(* CODESYS project sms_festo_lib_v1_1.library
   Company: Festo
   Description: 1.1.0 Added Intermediate Block
   Version: 1.1.0
   Placeholder: SMS Festo Lib V1.1
   Author: AJAY
   Title: SMS Festo Lib

Project tree, tasks and I/O mapping:
  libraries: Festo_CPX_API_EC_Beckhoff, * (Festo); Tc2_Standard, * (Beckhoff Automation GmbH); Tc2_System, * (Beckhoff Automation GmbH); Tc3_Module, * (Beckhoff Automation GmbH)
  DUTs/
    data type aByte_as_real
    data type UDT_ISDU_Command
    data type UDT_ReadParameter
    data type UDT_WriteParameter
  GVLs/
    global variables GVL
  POUs/
    function block SMS_Festo_Advanced [ST]
    function block SMS_Festo_Basic [ST]
    function block SMS_Festo_Intermediate [ST]
    function block SMS_Festo_IO [ST]
  Project Information/
    function F_GetCompany [ST]
    function F_GetTitle [ST]
    function F_GetVersion [ST]
  Version/
    global variables Global_Version
  VISUs/
*)

// DUTs/aByte_as_real
TYPE aByte_as_real :
UNION
	rRealValue: REAL;
	abyte: ARRAY  [0..3] OF BYTE;
END_UNION
END_TYPE

// DUTs/UDT_ISDU_Command
TYPE UDT_ISDU_Command :
STRUCT
	Net_Id: STRING;
	Ethercat_Address: 	UINT;
	Slot_Number: 	UINT;
	Port_Number: 	USINT;
	Para_Index: 	UINT;
	Para_SubIndex: 	USINT;
	Para_Length: 	UINT;
	Para_Data: 		ARRAY[0..231] OF BYTE;
	
END_STRUCT
END_TYPE

// DUTs/UDT_ReadParameter
TYPE UDT_ReadParameter :
STRUCT
	Index	:	UINT;	// Read Data Parameter Index Value
	Sub_index	:	USINT;	// Read Data Parameter Sub index Value
	Length		:	UINT;	// Read Data Parameter Length Value
	Value		:	DINT;	// Read Data Parameter Feedback Value
END_STRUCT
END_TYPE

// DUTs/UDT_WriteParameter
TYPE UDT_WriteParameter :
STRUCT
	Index		:	UINT;	// Send Data Parameter Index Value
	Sub_index		:	USINT;	// Send Data Parameter sub index Value
	Length			:	UINT;	// Send Data Parameter Length Value
	Value			:	DINT;	// Send Data Parameter Write Value
	NeedAction		:	BOOL;	// Send Data Parameter Need Action Decision 
	PreviousValue	:	DINT;	// Send Data Parameter Previous Write Value
	REAL_Value		:	REAL;	// Send Data Parameter Write REAL Value
END_STRUCT
END_TYPE

// GVLs/GVL
{attribute 'qualified_only'}
VAR_GLOBAL
	Inputs AT %I*: BYTE;
	Outputs AT %Q*: BYTE;
END_VAR

// Version/Global_Version
{attribute 'TcGenerated'}
{attribute 'no-analysis'}
{attribute 'linkalways'}
// This function has been automatically generated from the project information.
VAR_GLOBAL CONSTANT
	{attribute 'const_non_replaced'}
	stLibVersion_SMS_Festo_Lib : ST_LibVersion := (iMajor := 1, iMinor := 1, iBuild := 0, iRevision := 0, nFlags := 0, sVersion := '1.1.0');
END_VAR

// POUs/SMS_Festo_Advanced
FUNCTION_BLOCK SMS_Festo_Advanced
VAR_INPUT
	RefINPUTS: BYTE;					//Input Channel Mapping
	xEnable: BOOL; 						//True - Enable AOI function
	sNetId              : STRING;
	uiEthercatAddress   : UINT;          //Address of the slave device i.e. CPX-AP-I-EC-M12 Module
	uiSlotNumber        : UINT;          //Slot number where the IO Link master CPX-AP-I-4IOL-M12 module is connected
	usiPort             : USINT;          //Port of the CPX-AP-I-4IOL-M12 module where IO link device is connected
	xMoveIN: BOOL;						//TRUE - SMS moves inwards | FALSE - SMS Stops		
	xMoveIntermediate: BOOL;			//TRUE – SMS Moves to Intermediate Position | FALSE – SMS Stops
	xMoveOut: BOOL;						//TRUE - SMS moves outwards | FALSE - SMS Stops
	xQuitError: BOOL;					//TRUE - Reset Error Messages
	xPowerSMS: BOOL;					//TRUE - Enable power stage of SMS
	xUserInterfaceLock: BOOL;			//TRUE - lock user interface of SMS control unit
	bySpeedOut: BYTE := 1;				//Axix Move Speed Towards Out Direction 1 - 10% (default) | Limit 1 to 10
	bySpeedIN: BYTE:= 1;				//Axix Move Speed Towards IN Direction 1 - 10% (default) | Limit 1 to 10
	byForce: BYTE:= 1;					//Axix Move Force 1 - 10% (default) | Limit 1 to 10
	xReferenceDirection: BOOL;			//TRUE - Motor averted | FALSE - Motor side
	xExecuteReference: BOOL;			//TRUE – Start Homing
	diStartPressPosition: DINT:= 100;	//Defines Start Position of Stroke
	diIntermediatePosition: DINT:= 200;	//Defines Intermediate Position of Stroke
	diEndPosition: DINT:= 300;			//Defines End Position of Stroke
	xAutoStoreActive: BOOL;				//TRUE – Automatically stores the last downloaded parameters in the SMS.
	xStoreParameters: BOOL;				//TRUE – Manually stores the last downloaded parameters in the SMS.
	xReadDiagnosticData: BOOL;			//TRUE - Update value of outputs: O_DDTemperature, O_DDCurrent, O_DDVoltage, O_DDCyclesTotal, O_DDCyclesSinceReset, O_DDMileageTotal, O_DDMileageSinceReset
	xResetCounterMileage: BOOL;			//TRUE - Resets values of parameters “O_DDCyclesSinceReset”
	
END_VAR
VAR_OUTPUT
	RefOUTPUTS: BYTE;					//Output Channel Mapping
	xEnabled: BOOL;						//TRUE - AOI Function Enabled
	xWriteActive: BOOL;					//TRUE - Executing Parameter Write Function
	xWriteDone: BOOL;					//TRUE - Last Parameter Wrote Successful
	xReadActive: BOOL;					//TRUE - Parameter Read Function is Active
	xStateIn: BOOL;						//TRUE - SMS Axis Reached IN Position
	xStateIntermediate: BOOL;			//TRUE - SMS Axis Reached Intermediate Position
	xStateOut: BOOL;					//TRUE - SMS Axis Reached OUT Position
	xStateMove: BOOL;					//TRUE – SMS Axis at Moving Condition | FALSE – SMS Axis at Ideal Condition
	xError: BOOL;						//TRUE - SMS Module or AOI in Error State. Check Error Code
	uiLocalError: UINT;					//Function Block Local Error Code
	aErrorCode: ARRAY[0..15] OF WORD;	//SMS Error Code List
	diCurrentPosition: DINT;			//Axis Current Position Feedback
	diCurrentSpeed: DINT;				//Axis Current Speed Feedback
	diCurrentForce: DINT;				//Axis Current Force Feedback
	diDDTemprature: DINT;				//SMS Module Current Temperature Feedback
	diDDCurrent: DINT;					//SMS Module Present Value of Current
	diDDVoltage: DINT;					//SMS Module Present Voltage Feedback
	diDDCyclesTotal: DINT;				//Sum Value of Total Number of Axis Movement Cycle Count
	diDDCyclesSinceReset: DINT;			//Number of Axis Movement Cycle Count Since Reset Command
	diDDMileageTotal: DINT;				//Total Number of Movement Cycle in Engineering Unit
	diDDMileagesSinceReset: DINT;		//Number of Axis Movement Engineered Value Since Reset Command
	diNumOfStorageOperation: DINT;		//Total Number of Auto Store Operation Done Sofare
	
END_VAR

VAR
	Lt_ReadParaData: ARRAY[0..19] OF UDT_ReadParameter;
	Lt_WriteParaData: ARRAY[0..19] OF UDT_WriteParameter;
	Lt_ErrorRawData: ARRAY [0..48] OF BYTE;
	Lt_RiseEdgePowerSMS: BOOL;
	Lt_FalingEdgePowerSMS: BOOL;
	Lt_RiseUserInterfaceLock: BOOL;
	Lt_FalingEdgeUserInterfaceLock: BOOL;
	Lt_RiseReferenceDirection: BOOL;
	Lt_FalingEdgeReferenceDirection: BOOL;
	Lt_RiseExecuteReference: BOOL;
	Lt_FalingEdgeExecuteReference: BOOL;
	Lt_RiseStoreParameters: BOOL;
	Lt_FalingEdgeStoreParameters: BOOL;
	Lt_RiseResetCounterMileage: BOOL;
	Lt_FalingEdgeResetCounterMileage: BOOL;
	Lt_RiseAutoStoreActive: BOOL;
	Lt_FalingEdgeAutoStoreActive: BOOL;
	Lt_RiseEnableFileHandling: BOOL;
	Lt_FalingEdgeEnableFileHandling: BOOL;
	Step_SEQ: INT;
	Lt_ReadIndex: INT;
	Lt_WriteIndex: INT;
	Lt_Read_Parameter_ISDU: UDT_ISDU_Command;
	Lt_Write_Parameter_ISDU: UDT_ISDU_Command;
	Lt_ForLength: INT;
	Lt_Execute_Read: BOOL;
	Lt_Execute_Write: BOOL; 
	Lt_StateDevice: BOOL;
	Lt_ScanCount: DINT;
	Lt_ScanCount02: DINT;
	Lt_ScanCount03: DINT;
	Lt_ScanCount001: DINT;
	Lt_DeviceState_RisingEdge: BOOL;
	Lt_RealConvert: aByte_as_real;
	Lt_ExecuteReference_RisingEdge: BOOL;
	Lt_ExecuteReference_Trigger: BOOL;
	Lt_ExecuteReference_Trigger01: BOOL;	
	Lt_IsItString: BOOL;
	Lt_Startposition: REAL;
	Lt_Intermediateposition: REAL;
	Lt_Endposition: REAL;
	Lt_ReCurrentPosition: REAL;
	Lt_ReCurrentPosition1: DINT;
	LT_ParameterRewriteDelay: BOOL;
	Lt_ExecuteReference_Trigger02: BOOL;
	Lt_NumOfStorageOperation:Dint;
	
	ReadPara: CPXAPI_IOLink_Parameter;
	WritePara: CPXAPI_IOLink_Parameter;
	Delay_Timmer: TON;
	Elapse_time: TIME;
END_VAR

(*
fkjhfkjsdhjkfhsdjkfhkjhhh
jdhfjkdhjkfhdkjhf
*)

(*
===============================================================================================================
Advice TO Released Library Revisions 
===============================================================================================================
SMS_Festo_Lib | Communication: Beckhoff EtherCat
---------------------------------------------------------------------------------------------------------------
Version                           Date of Release
V1.0                                07.01.2022
V1.1                                03.06.2022

---------------------------------------------------------------------------------------------------------------
Changes in Library:

V1.0 -  Release Version


V1.1 - Position variables datatype changed from Real to Dint.
       Autostorage parameter continuous count bug fixed.
       Number of storage parameter double count bug fixed. 
*)

// Enable Function Block Sequence Logic------------------------------------------------------------------------ 
IF xEnable THEN 				
	xEnabled					:= TRUE;
	
ELSE
	xEnabled					:= FALSE;
	xWriteActive				:= FALSE;	
	xWriteDone					:= FALSE;
	xReadActive					:= FALSE;
	Step_SEQ					:= 0;
	Lt_ReadParaData[0].Value	:= 0;
	Lt_ReadParaData[1].Value	:= 0;
	Lt_ReadParaData[2].Value	:= 0;
	Lt_ReadParaData[3].Value	:= 0;
	Lt_ReadParaData[4].Value	:= 0;
	Lt_ReadParaData[5].Value	:= 0;
	Lt_ReadParaData[6].Value	:= 0;
	Lt_ReadParaData[7].Value	:= 0;
	Lt_ReadParaData[8].Value	:= 0;
	Lt_ReadParaData[9].Value	:= 0;
	Lt_ReadParaData[10].Value	:= 0;
	Lt_ReadParaData[11].Value	:= 0;
	
END_IF

//Process Data Command Logic---------------------------------------------------------------------------------------
IF xEnabled THEN				
	
	IF xMoveIN THEN				// Move IN Position Command
		RefOUTPUTS.0	:= TRUE;
	ELSE
		RefOUTPUTS.0	:= FALSE;
	END_IF
	
	IF xMoveOut THEN			// Move OUT Position Command
		RefOUTPUTS.1	:= TRUE;
	ELSE
		RefOUTPUTS.1	:= FALSE;	
	END_IF
	
	IF xMoveIntermediate THEN	// Move Intermediat Position Command
		RefOUTPUTS.4	:= TRUE;
	ELSE
		RefOUTPUTS.4	:= FALSE;	
	END_IF
	
	IF xQuitError THEN			// Move Quite Error Command
		RefOUTPUTS.2	:= TRUE;
	ELSE
		RefOUTPUTS.2	:= FALSE;	
	END_IF
ELSE							// Clear Command When FB Not Enabled
	RefOUTPUTS.0	:= FALSE;	
	RefOUTPUTS.1	:= FALSE;	
	RefOUTPUTS.2	:= FALSE;
	RefOUTPUTS.4	:= FALSE;
END_IF


// Process Data Feedback Logic---------------------------------------------------------------------------------
IF xEnabled THEN				
	
	IF RefINPUTS.0 THEN				// IN Position Status
		xStateIn	:= TRUE;
	ELSE
		xStateIn	:= FALSE;
	END_IF
	
	IF RefINPUTS.1 THEN				// Out Position Status
		xStateOut	:= TRUE;
	ELSE
		xStateOut	:= FALSE;
	END_IF
	
	IF RefINPUTS.2 THEN				// Axis Moving Status
		xStateMove	:= TRUE;
	ELSE
		xStateMove	:= FALSE;
	END_IF
	
	IF RefINPUTS.3 THEN				// Device Healthy Status
		Lt_StateDevice	:= TRUE;
	ELSE
		Lt_StateDevice	:= FALSE;
	END_IF
	
	IF RefINPUTS.4 THEN				// Intermediat Position Status
		xStateIntermediate	:= TRUE;
	ELSE
		xStateIntermediate	:= FALSE;
	END_IF	
ELSE 								// Clear Status When FB is Not Enabled
	xStateIn			:= FALSE;
	xStateOut			:= FALSE;
	xStateMove			:= FALSE;
	xStateIntermediate	:= FALSE;
	Lt_StateDevice		:= FALSE;
END_IF

// Device Error State Logic -----------------------------------------------------------------------------------
IF xEnabled AND xStateIn AND xStateOut AND NOT Lt_StateDevice THEN
	xError	:= TRUE;
ELSE
	xError	:= FALSE;
END_IF

// After Homing Parameters Re-Write Logic ---------------------------------------------------------------------
IF Lt_ExecuteReference_Trigger01	AND NOT xStateMove THEN
	Lt_ExecuteReference_Trigger02:= TRUE;
	
	IF LT_ParameterRewriteDelay THEN
		Lt_WriteParaData[0].PreviousValue	:= 0;
		Lt_WriteParaData[1].PreviousValue	:= 0;
		Lt_WriteParaData[2].PreviousValue	:= 0;
		Lt_WriteParaData[3].PreviousValue	:= 0;
		Lt_WriteParaData[4].PreviousValue	:= 0;
		Lt_WriteParaData[5].PreviousValue	:= 0;
		Lt_WriteParaData[7].PreviousValue	:= 0;
		Lt_WriteParaData[8].PreviousValue	:= 0;
		Lt_WriteParaData[12].PreviousValue	:= 0;
		Lt_ExecuteReference_Trigger01		:= FALSE;
		Lt_ExecuteReference_Trigger02		:= FALSE;
		
	END_IF
ELSE
		Lt_ExecuteReference_Trigger02		:= FALSE;
END_IF
// After Homing Parameter Rewrite Delay
Delay_Timmer(IN:= Lt_ExecuteReference_Trigger02, PT:=T#6S , Q=> LT_ParameterRewriteDelay, ET=> Elapse_time );

//Setpoint Limit Error-----------------------------------------------------------------------------------------
IF (bySpeedIN < 1 ) OR (bySpeedIN > 10 ) THEN 
	uiLocalError := 1001;
	xError		 := TRUE;

ELSIF (bySpeedOut < 1 ) OR (bySpeedOut > 10 ) THEN
	uiLocalError := 1002;
	xError		 := TRUE;
ELSIF (bySpeedIN < 1 ) OR (bySpeedIN > 10 ) THEN
	uiLocalError := 1003;
	xError		 := TRUE;
END_IF

//Device Status Rising Edge Logic--------------------------------------------------------------------------------
IF Lt_StateDevice AND NOT Lt_DeviceState_RisingEdge THEN
	Lt_DeviceState_RisingEdge	:= TRUE;
	xError						:= FALSE;
ELSIF NOT Lt_StateDevice THEN
	Lt_DeviceState_RisingEdge	:= FALSE;
END_IF

//Execute Ref Rising Edge Logic--------------------------------------------------------------------------------
IF xExecuteReference AND NOT Lt_ExecuteReference_RisingEdge THEN
	Lt_ExecuteReference_RisingEdge	:= TRUE;
	Lt_ExecuteReference_Trigger		:= TRUE;
	xError							:= FALSE;
ELSIF NOT xExecuteReference THEN
	Lt_ExecuteReference_RisingEdge	:= FALSE;
END_IF

// Quite Error Logic ------------------------------------------------------------------------------------------
IF xQuitError AND xEnabled THEN
	Step_SEQ			:= 0;
	xWriteActive		:= FALSE;
	xWriteDone			:= FALSE;
	xReadActive			:= FALSE;
	xError				:= FALSE;
	uiLocalError		:= 0;	
	
	// Clear Error Data Raw Array
		
				Lt_ErrorRawData[0] 		:= 0; Lt_ErrorRawData[1] 	:= 0; Lt_ErrorRawData[2] 	:= 0; Lt_ErrorRawData[3] 	:= 0;
				Lt_ErrorRawData[4] 		:= 0; Lt_ErrorRawData[5] 	:= 0; Lt_ErrorRawData[6] 	:= 0; Lt_ErrorRawData[7] 	:= 0;
				Lt_ErrorRawData[8] 		:= 0; Lt_ErrorRawData[9] 	:= 0; Lt_ErrorRawData[10] 	:= 0; Lt_ErrorRawData[11] 	:= 0;
				Lt_ErrorRawData[12] 	:= 0; Lt_ErrorRawData[13] 	:= 0; Lt_ErrorRawData[14] 	:= 0; Lt_ErrorRawData[15] 	:= 0;
				Lt_ErrorRawData[16] 	:= 0; Lt_ErrorRawData[17] 	:= 0; Lt_ErrorRawData[18] 	:= 0; Lt_ErrorRawData[19] 	:= 0;
				Lt_ErrorRawData[20] 	:= 0; Lt_ErrorRawData[21] 	:= 0; Lt_ErrorRawData[22] 	:= 0; Lt_ErrorRawData[23] 	:= 0;
				Lt_ErrorRawData[24] 	:= 0; Lt_ErrorRawData[25] 	:= 0; Lt_ErrorRawData[26] 	:= 0; Lt_ErrorRawData[27] 	:= 0;
				Lt_ErrorRawData[28] 	:= 0; Lt_ErrorRawData[29] 	:= 0; Lt_ErrorRawData[30] 	:= 0; Lt_ErrorRawData[31] 	:= 0;
				Lt_ErrorRawData[32] 	:= 0; Lt_ErrorRawData[33] 	:= 0; Lt_ErrorRawData[34] 	:= 0; Lt_ErrorRawData[35] 	:= 0;
				Lt_ErrorRawData[36] 	:= 0; Lt_ErrorRawData[37] 	:= 0; Lt_ErrorRawData[38] 	:= 0; Lt_ErrorRawData[39] 	:= 0;
				Lt_ErrorRawData[40] 	:= 0; Lt_ErrorRawData[41] 	:= 0; Lt_ErrorRawData[42] 	:= 0; Lt_ErrorRawData[43] 	:= 0;
				Lt_ErrorRawData[44] 	:= 0; Lt_ErrorRawData[45] 	:= 0; Lt_ErrorRawData[46] 	:= 0; Lt_ErrorRawData[47] 	:= 0;
				Lt_ErrorRawData[48] 	:= 0;		
END_IF

//Power Stage Enable & Disable Command Write Input Parameter Logic----------------------------------------------
IF xPowerSMS AND NOT Lt_RiseEdgePowerSMS THEN
	Lt_WriteParaData[0].NeedAction	:= TRUE;
	Lt_RiseEdgePowerSMS				:=	TRUE;
	Lt_FalingEdgePowerSMS			:=	FALSE;
	Lt_WriteParaData[0].Value		:= 16#0CC;
	
ELSIF NOT xPowerSMS	AND NOT Lt_FalingEdgePowerSMS THEN
	Lt_WriteParaData[0].NeedAction	:= TRUE;
	Lt_RiseEdgePowerSMS				:=	FALSE;
	Lt_FalingEdgePowerSMS			:=	TRUE;
	Lt_WriteParaData[0].Value		:= 16#0CB;
END_IF;


Lt_WriteParaData[0].Index		:= 2;
Lt_WriteParaData[0].Length			:= 1;
Lt_WriteParaData[0].Sub_index		:= 0;

//User Interface Lock Command Write Parameter Logic------------------------------------------------------------- 
IF xUserInterfaceLock AND NOT Lt_RiseUserInterfaceLock THEN
	Lt_WriteParaData[1].NeedAction	:= TRUE;
	Lt_RiseUserInterfaceLock 		:= TRUE;
	Lt_FalingEdgeUserInterfaceLock	:= FALSE;
	Lt_WriteParaData[1].Value		:= 1;
	
ELSIF NOT xUserInterfaceLock	AND NOT Lt_FalingEdgeUserInterfaceLock THEN
	Lt_WriteParaData[1].NeedAction	:= TRUE;
	Lt_RiseUserInterfaceLock		:= FALSE;
	Lt_FalingEdgeUserInterfaceLock	:= TRUE;
	Lt_WriteParaData[1].Value		:= 0;
END_IF;


Lt_WriteParaData[1].Index		:= 16#000C;
Lt_WriteParaData[1].Length			:= 1;
Lt_WriteParaData[1].Sub_index		:= 16#4;

//Speed Out % Command Write Parameter Logic--------------------------------------------------------------------- 
IF Lt_WriteParaData[2].Value <> Lt_WriteParaData[2].PreviousValue THEN 
	Lt_WriteParaData[2].NeedAction	:= TRUE;	
ELSE
	Lt_WriteParaData[2].NeedAction	:= FALSE;
	
END_IF

Lt_WriteParaData[2].Value			:= bySpeedOut;
Lt_WriteParaData[2].Sub_index		:= 16#0;
Lt_WriteParaData[2].Index		:= 16#101;
Lt_WriteParaData[2].Length			:= 1;


//Speed IN % Command Write Parameter Logic---------------------------------------------------------------------- 
IF Lt_WriteParaData[3].Value <> Lt_WriteParaData[3].PreviousValue THEN 
	Lt_WriteParaData[3].NeedAction	:= TRUE;	
ELSE
	Lt_WriteParaData[3].NeedAction	:= FALSE;
END_IF

Lt_WriteParaData[3].Value			:= bySpeedIN;
Lt_WriteParaData[3].Sub_index		:= 16#0;
Lt_WriteParaData[3].Index		:= 16#100;
Lt_WriteParaData[3].Length			:= 1;


//Force % Command Write Parameter Logic------------------------------------------------------------------------ 
IF Lt_WriteParaData[4].Value <> Lt_WriteParaData[4].PreviousValue THEN 
	Lt_WriteParaData[4].NeedAction	:= TRUE;	
ELSE
	Lt_WriteParaData[4].NeedAction	:= FALSE;
END_IF

Lt_WriteParaData[4].Value			:= byForce;
Lt_WriteParaData[4].Sub_index		:= 16#0;
Lt_WriteParaData[4].Index		:= 16#102;
Lt_WriteParaData[4].Length			:= 1;


//Referance Direction Command Write Parameter Logic----------------------------------------------------------- 
IF xReferenceDirection AND NOT Lt_RiseReferenceDirection THEN
	Lt_WriteParaData[5].NeedAction	:= TRUE;
	Lt_RiseReferenceDirection 		:= TRUE;
	Lt_FalingEdgeReferenceDirection	:= FALSE;
	Lt_WriteParaData[5].Value		:= 1;
	
ELSIF NOT xReferenceDirection	AND NOT Lt_FalingEdgeReferenceDirection THEN
	Lt_WriteParaData[5].NeedAction	:= TRUE;
	Lt_RiseReferenceDirection 		:= FALSE;
	Lt_FalingEdgeReferenceDirection	:= TRUE;
	Lt_WriteParaData[5].Value		:= 0;
END_IF;


Lt_WriteParaData[5].Index		:= 16#103;
Lt_WriteParaData[5].Length			:= 1;
Lt_WriteParaData[5].Sub_index		:= 16#0;

//Execute Referance Command | Write Parameter Logic------------------------------------------------------------ 
IF Lt_ExecuteReference_Trigger  THEN
	Lt_WriteParaData[6].NeedAction	:= TRUE;
	Lt_WriteParaData[6].Value		:= 1;
	Lt_ExecuteReference_Trigger		:= FALSE;
	Lt_ExecuteReference_Trigger01	:= TRUE;
		
ELSIF NOT xExecuteReference	 THEN
	Lt_WriteParaData[6].Value		:= 0;
END_IF;


Lt_WriteParaData[6].Index		:= 16#104;
Lt_WriteParaData[6].Length			:= 1;
Lt_WriteParaData[6].Sub_index		:= 16#0;

//Start Press Position Command | Write Parameter Logic---------------------------------------------------------- 
IF Lt_WriteParaData[12].Value <> Lt_WriteParaData[12].PreviousValue THEN 
	Lt_WriteParaData[12].NeedAction	:= TRUE;	
ELSE
	Lt_WriteParaData[12].NeedAction	:= FALSE;
END_IF

Lt_WriteParaData[12].REAL_Value		:= TO_REAL(diStartPressPosition);
Lt_WriteParaData[12].Value			:= diStartPressPosition;
Lt_WriteParaData[12].Sub_index		:= 16#0;
Lt_WriteParaData[12].Index		:= 16#105;
Lt_WriteParaData[12].Length			:= 4;


//End Position Command | Write Parameter Logic------------------------------------------------------------------- 
IF Lt_WriteParaData[7].Value <> Lt_WriteParaData[7].PreviousValue THEN 
	Lt_WriteParaData[7].NeedAction	:= TRUE;	
ELSE
	Lt_WriteParaData[7].NeedAction	:= FALSE;
END_IF
Lt_WriteParaData[7].REAL_Value		:= TO_REAL(diEndPosition);
Lt_WriteParaData[7].Value			:= diEndPosition;
Lt_WriteParaData[7].Sub_index		:= 16#0;
Lt_WriteParaData[7].Index		:= 16#106;
Lt_WriteParaData[7].Length			:= 4;


//Store Parameters Command | Write Parameter Logic--------------------------------------------------------------- 
IF xStoreParameters AND NOT Lt_RiseStoreParameters AND xEnabled THEN
	Lt_WriteParaData[9].NeedAction	:= TRUE;
	Lt_RiseStoreParameters 			:= TRUE;
	Lt_FalingEdgeStoreParameters	:= FALSE;
	Lt_WriteParaData[9].Value		:= 1;
	
ELSIF NOT xStoreParameters	AND NOT Lt_FalingEdgeStoreParameters AND xEnabled THEN
	Lt_WriteParaData[9].NeedAction	:= TRUE;
	Lt_RiseStoreParameters  		:= FALSE;
	Lt_FalingEdgeStoreParameters	:= TRUE;
	Lt_WriteParaData[9].Value		:= 0;
END_IF;


Lt_WriteParaData[9].Index		:= 16#10B;
Lt_WriteParaData[9].Length			:= 1;
Lt_WriteParaData[9].Sub_index		:= 16#0;

//Reset Counter Mileage Command | Write Parameter Logic ----------------------------------------------------------
IF xResetCounterMileage AND NOT Lt_RiseResetCounterMileage  THEN
	Lt_WriteParaData[10].NeedAction	:= TRUE;
	//Lt_WriteParaData[11].NeedAction	:= TRUE;
	Lt_RiseResetCounterMileage 		:= TRUE;
	Lt_FalingEdgeResetCounterMileage:= FALSE;
	Lt_WriteParaData[10].Value		:= 1;
	//Lt_WriteParaData[11].Value		:= 1;
	
ELSIF NOT xResetCounterMileage	AND NOT Lt_FalingEdgeResetCounterMileage  THEN
	Lt_WriteParaData[10].NeedAction	:= TRUE;
	
	Lt_RiseResetCounterMileage  	:= FALSE;
	Lt_FalingEdgeResetCounterMileage:= TRUE;
	Lt_WriteParaData[10].Value		:= 0;
	//Lt_WriteParaData[11].Value		:= 0;
END_IF;


Lt_WriteParaData[10].Index		:= 16#12A;
Lt_WriteParaData[10].Length			:= 1;
Lt_WriteParaData[10].Sub_index		:= 16#0;

Lt_WriteParaData[11].NeedAction	:= FALSE; // Array Number 11 Will be Dummy, So Always OFF (No Action)
//Lt_WriteParaData[11].IO_Link_Format	:= 0;
//Lt_WriteParaData[11].Instance		:= 16#12A;
//Lt_WriteParaData[11].Length			:= 4;
//Lt_WriteParaData[11].Attribute		:= 16#0;

//Intermediate Position Command | Write Parameter Logic ------------------------------------------------------------
IF Lt_WriteParaData[8].Value <> Lt_WriteParaData[8].PreviousValue THEN 
	Lt_WriteParaData[8].NeedAction	:= TRUE;	
ELSE
	Lt_WriteParaData[8].NeedAction	:= FALSE;
END_IF
Lt_WriteParaData[8].REAL_Value		:= TO_REAL(diIntermediatePosition);
Lt_WriteParaData[8].Value			:= diIntermediatePosition;
Lt_WriteParaData[8].Sub_index		:= 16#0;
Lt_WriteParaData[8].Index		:= 16#108;
Lt_WriteParaData[8].Length			:= 4;


//Auto Store Parameters Command | Write Parameter Logic------------------------------------------------------------- 
IF xAutoStoreActive AND NOT Lt_RiseAutoStoreActive  THEN
	Lt_WriteParaData[13].NeedAction	:= TRUE;
	Lt_RiseAutoStoreActive 			:= TRUE;
	Lt_FalingEdgeAutoStoreActive	:= FALSE;
	Lt_WriteParaData[13].Value		:= 1;
	
ELSIF NOT xAutoStoreActive	AND NOT Lt_FalingEdgeAutoStoreActive  THEN
	Lt_WriteParaData[13].NeedAction	:= TRUE;
	Lt_RiseAutoStoreActive  		:= FALSE;
	Lt_FalingEdgeAutoStoreActive	:= TRUE;
	Lt_WriteParaData[13].Value		:= 0;
END_IF;


Lt_WriteParaData[13].Index		:= 16#109;
Lt_WriteParaData[13].Length			:= 1;
Lt_WriteParaData[13].Sub_index		:= 16#0;

//Enable File Handling Parameters Command | Write Parameter Logic----------------------------------------------------
//IF xEnableFileHandling AND NOT Lt_RiseEnableFileHandling  THEN
//	Lt_WriteParaData[14].NeedAction	:= TRUE;
//	Lt_RiseEnableFileHandling		:= TRUE;
//	Lt_FalingEdgeEnableFileHandling	:= FALSE;
//	Lt_WriteParaData[14].Value		:= 8782;
	
//ELSIF NOT xEnableFileHandling	AND NOT Lt_FalingEdgeEnableFileHandling  THEN
//	Lt_WriteParaData[14].NeedAction	:= TRUE;
//	Lt_RiseEnableFileHandling  		:= FALSE;
//	Lt_FalingEdgeEnableFileHandling	:= TRUE;
//	Lt_WriteParaData[14].Value		:= 0;
//END_IF;

//Lt_WriteParaData[14].IO_Link_Format	:= 15;
//Lt_WriteParaData[14].Instance		:= 16#3000;
//Lt_WriteParaData[14].Length			:= 2;
//Lt_WriteParaData[14].Attribute		:= 16#0;

//Execute File Handling Parameters Command | Write Parameter Logic--------------------------------------------------
//Lt_WriteParaData[15].IO_Link_Format	:= 15;
//Lt_WriteParaData[15].Instance		:= 16#3001;
//Lt_WriteParaData[15].Length			:= 2;
//Lt_WriteParaData[15].Attribute		:= 16#0;
//Lt_WriteParaData[15].Value			:= xExecuteFileHandling;

//Read & Write Control Sequence Logic-------------------------------------------------------------------------------
CASE Step_SEQ OF 					
	0:	// Enable Read & Write Logic
		IF xEnabled THEN 
			Lt_ReadIndex	:= 0;
			Lt_WriteIndex	:= 0;
			Step_SEQ		:= 10;
		ELSE
			Step_SEQ		:= 0;
		END_IF
	10:	// Read Data Parameter Input Logic 
		Lt_Read_Parameter_ISDU.Net_Id	        :=	sNetId ;
		Lt_Read_Parameter_ISDU.Ethercat_Address	:=	uiEthercatAddress ;
		Lt_Read_Parameter_ISDU.Slot_Number	    :=	uiSlotNumber ;
		Lt_Read_Parameter_ISDU.Port_Number		:=	usiPort;
		Lt_Read_Parameter_ISDU.Para_Index		:=	Lt_ReadParaData[Lt_ReadIndex].Index;
		Lt_Read_Parameter_ISDU.Para_SubIndex	:=	Lt_ReadParaData[Lt_ReadIndex].Sub_index;
		Lt_Read_Parameter_ISDU.Para_Length		:=	Lt_ReadParaData[Lt_ReadIndex].Length;
		Lt_Read_Parameter_ISDU.Para_Data[0]		:=	0;
		Lt_Read_Parameter_ISDU.Para_Data[1]		:=	0;
		Lt_Read_Parameter_ISDU.Para_Data[2]		:=	0;
		Lt_Read_Parameter_ISDU.Para_Data[3]		:=	0;
		
		IF (Lt_ReadIndex = 3)	THEN	// Is It String Command Mapping for Read Instruction 
			Lt_IsItString	:= TRUE;
			ELSE 
			Lt_IsItString	:= FALSE;
		END_IF
		
		
		xReadActive						:= TRUE;
		xWriteActive					:= FALSE;
		Step_SEQ						:= 20;
		
	20:	// Read Command Enable Logic 
		
			Lt_Execute_Read		:=	TRUE;	 
		 	Step_SEQ			:= 21;
			
	21: // Read Feedback Data Manipulation
		IF ReadPara.xDone	THEN
			
			IF Lt_ReadIndex <> 3 THEN
				Lt_ForLength	:= 0;
				IF 	(Lt_ReadParaData[Lt_ReadIndex].Length = 4) THEN
					Lt_ReadParaData[Lt_ReadIndex].Value	:= TO_DINT(Lt_Read_Parameter_ISDU.Para_Data[0]) + SHL(TO_DINT(Lt_Read_Parameter_ISDU.Para_Data[1]),8)	+ SHL(TO_DINT(Lt_Read_Parameter_ISDU.Para_Data[2]),16) 
														+ SHL(TO_DINT(Lt_Read_Parameter_ISDU.Para_Data[3]),24);
														
				ELSIF (Lt_ReadParaData[Lt_ReadIndex].Length = 2) THEN
					Lt_ReadParaData[Lt_ReadIndex].Value	:= TO_DINT(Lt_Read_Parameter_ISDU.Para_Data[0]) + SHL(TO_DINT(Lt_Read_Parameter_ISDU.Para_Data[1]),8);
			
				ELSIF (Lt_ReadParaData[Lt_ReadIndex].Length = 1) THEN
					Lt_ReadParaData[Lt_ReadIndex].Value	:= TO_DINT(Lt_Read_Parameter_ISDU.Para_Data[0]);
				END_IF;
					
			ELSE
			
				Lt_ErrorRawData[0] 		:= ReadPara.pData[0];	 Lt_ErrorRawData[1] := ReadPara.pData[1]; 	Lt_ErrorRawData[2] 	:= ReadPara.pData[2]; Lt_ErrorRawData[3] 	:= ReadPara.pData[3];
				Lt_ErrorRawData[4] 		:= ReadPara.pData[4]; 	Lt_ErrorRawData[5] 	:= ReadPara.pData[5];	Lt_ErrorRawData[6] 	:= ReadPara.pData[6]; Lt_ErrorRawData[7] 	:= ReadPara.pData[7];
				Lt_ErrorRawData[8] 		:= ReadPara.pData[8]; 	Lt_ErrorRawData[9] 	:= ReadPara.pData[9]; 	Lt_ErrorRawData[10] := ReadPara.pData[10]; Lt_ErrorRawData[11] 	:= ReadPara.pData[11];
				Lt_ErrorRawData[12] 	:= ReadPara.pData[12]; Lt_ErrorRawData[13] 	:= ReadPara.pData[13]; Lt_ErrorRawData[14] 	:= ReadPara.pData[14]; Lt_ErrorRawData[15] 	:= ReadPara.pData[15];
				Lt_ErrorRawData[16] 	:= ReadPara.pData[16]; Lt_ErrorRawData[17] 	:= ReadPara.pData[17]; Lt_ErrorRawData[18] 	:= ReadPara.pData[18]; Lt_ErrorRawData[19] 	:= ReadPara.pData[19];
				Lt_ErrorRawData[20] 	:= ReadPara.pData[20]; Lt_ErrorRawData[21] 	:= ReadPara.pData[21]; Lt_ErrorRawData[22] 	:= ReadPara.pData[22]; Lt_ErrorRawData[23] 	:= ReadPara.pData[23];
				Lt_ErrorRawData[24] 	:= ReadPara.pData[24]; Lt_ErrorRawData[25] 	:= ReadPara.pData[25]; Lt_ErrorRawData[26] 	:= ReadPara.pData[26]; Lt_ErrorRawData[27] 	:= ReadPara.pData[27];
				Lt_ErrorRawData[28] 	:= ReadPara.pData[28]; Lt_ErrorRawData[29] 	:= ReadPara.pData[29]; Lt_ErrorRawData[30] 	:= ReadPara.pData[30]; Lt_ErrorRawData[31] 	:= ReadPara.pData[31];
				Lt_ErrorRawData[32] 	:= ReadPara.pData[32]; Lt_ErrorRawData[33] 	:= ReadPara.pData[33]; Lt_ErrorRawData[34] 	:= ReadPara.pData[34]; Lt_ErrorRawData[35] 	:= ReadPara.pData[35];
				Lt_ErrorRawData[36] 	:= ReadPara.pData[36]; Lt_ErrorRawData[37] 	:= ReadPara.pData[37]; Lt_ErrorRawData[38] 	:= ReadPara.pData[38]; Lt_ErrorRawData[39] 	:= ReadPara.pData[39];
				Lt_ErrorRawData[40] 	:= ReadPara.pData[40]; Lt_ErrorRawData[41] 	:= ReadPara.pData[41]; Lt_ErrorRawData[42] 	:= ReadPara.pData[42]; Lt_ErrorRawData[43] 	:= ReadPara.pData[43];
				Lt_ErrorRawData[44] 	:= ReadPara.pData[44]; Lt_ErrorRawData[45] 	:= ReadPara.pData[45]; Lt_ErrorRawData[46] 	:= ReadPara.pData[46]; Lt_ErrorRawData[47] 	:= ReadPara.pData[47];
				Lt_ErrorRawData[48] 	:= ReadPara.pData[48];
			
			END_IF
			
			Lt_ScanCount03	:= Lt_ScanCount03 + 1;
			IF Lt_ScanCount03 > 2 THEN 
			Lt_Execute_Read					:= FALSE;
			Step_SEQ						:= 30;
			Lt_ScanCount03					:= 0;
			END_IF
			
		ELSIF	ReadPara.xError	THEN 
			
			uiLocalError					:= 1004;
			Lt_Execute_Read					:= FALSE;
			Step_SEQ						:= 999;
			
		END_IF
	30:	// Read Parameter List Index & Move Sequence to Write Function Logic
		IF ( Lt_ReadIndex <= 11 ) THEN
			
			Lt_ReadIndex 	:= Lt_ReadIndex + 1;
			Step_SEQ		:= 10;
		END_IF 
		
		IF ( xReadDiagnosticData AND Lt_ReadIndex >= 12 ) OR ( NOT xReadDiagnosticData AND Lt_ReadIndex >= 4 ) THEN
			
			Lt_WriteIndex	:= 0;
			Step_SEQ		:= 35;
			
		END_IF
		
	35:
			Lt_Write_Parameter_ISDU.Para_Data[0]	:= 0;	
			Lt_Write_Parameter_ISDU.Para_Data[1]	:= 0;
			Lt_Write_Parameter_ISDU.Para_Data[2]	:= 0;
			Lt_Write_Parameter_ISDU.Para_Data[3]	:= 0;	
			Step_SEQ								:= 40;
			
	40:	// Write Data Parameter Input Logic 
		Lt_Write_Parameter_ISDU.Net_Id	:=	sNetId;
		Lt_Write_Parameter_ISDU.Ethercat_Address	:=	uiEthercatAddress;
		Lt_Write_Parameter_ISDU.Slot_Number	:=	uiSlotNumber;
		Lt_Write_Parameter_ISDU.Port_Number	:=	usiPort;
		Lt_Write_Parameter_ISDU.Para_Index	:=	Lt_WriteParaData[Lt_WriteIndex].Index;
		Lt_Write_Parameter_ISDU.Para_SubIndex	:=	Lt_WriteParaData[Lt_WriteIndex].Sub_index;
		Lt_Write_Parameter_ISDU.Para_Length	:=	Lt_WriteParaData[Lt_WriteIndex].Length;
		
		IF Lt_Write_Parameter_ISDU.Para_Length = 4 THEN
			
			Lt_RealConvert.rRealValue				:= Lt_WriteParaData[Lt_WriteIndex].REAL_Value;
			Lt_Write_Parameter_ISDU.Para_Data[0]	:= Lt_RealConvert.abyte[0];	
			Lt_Write_Parameter_ISDU.Para_Data[1]	:= Lt_RealConvert.abyte[1];
			Lt_Write_Parameter_ISDU.Para_Data[2]	:= Lt_RealConvert.abyte[2];
			Lt_Write_Parameter_ISDU.Para_Data[3]	:= Lt_RealConvert.abyte[3];	
		
		ELSIF Lt_Write_Parameter_ISDU.Para_Length = 2 THEN
			Lt_Write_Parameter_ISDU.Para_Data[0]	:=	TO_BYTE(Lt_WriteParaData[Lt_WriteIndex].Value);
			Lt_Write_Parameter_ISDU.Para_Data[1]	:=	TO_BYTE(SHR(Lt_WriteParaData[Lt_WriteIndex].Value,8));
		
		ELSIF Lt_Write_Parameter_ISDU.Para_Length = 1 THEN
			Lt_Write_Parameter_ISDU.Para_Data[0]	:=	TO_BYTE(Lt_WriteParaData[Lt_WriteIndex].Value);
		END_IF
		
		Lt_ScanCount	:= Lt_ScanCount + 1;
		
		IF 	Lt_ScanCount >= 2 THEN
		xReadActive						:= FALSE;
		//xWriteActive					:= TRUE;
		Lt_ScanCount					:= 0;	
		Step_SEQ						:= 50;
		END_IF
	
	50:	// Write Command Enable Logic 
		IF Lt_WriteIndex <> 7 THEN
            IF Lt_WriteParaData[Lt_WriteIndex].NeedAction THEN
                Lt_Execute_Write := TRUE;
                xWriteDone := FALSE;
				xReadActive	:= FALSE;
		        xWriteActive:= TRUE;
                Step_SEQ := 51;
            ELSE
                Step_SEQ := 60;
            END_IF;
        ELSE
            IF NOT Lt_ExecuteReference_Trigger01 THEN
                IF Lt_WriteParaData[Lt_WriteIndex].NeedAction THEN
                    Lt_Execute_Write := TRUE;
                    xWriteDone := FALSE;
					xReadActive	:= FALSE;
		            xWriteActive:= TRUE;
                    Step_SEQ := 51;
                ELSE
                    Step_SEQ := 60;
                END_IF;
            END_IF;
        END_IF;
				
	51:	// Write Data Manipulation
		IF WritePara.xDone THEN
			Lt_WriteParaData[Lt_WriteIndex].NeedAction		:= FALSE;
			Lt_WriteParaData[Lt_WriteIndex].PreviousValue	:= Lt_WriteParaData[Lt_WriteIndex].Value;
			Lt_Execute_Write								:= FALSE;
			xWriteDone										:= TRUE;
			xWriteActive									:= FALSE;
			Step_SEQ										:= 60;	 
		ELSIF WritePara.xError	THEN
			uiLocalError		:= 1005;
			Lt_Execute_Write	:= FALSE;
			Step_SEQ			:= 999;
		 END_IF
	
	60:	// Write Parameter List Index & Move Sequence to Read Function Logic
		IF ( Lt_WriteIndex <= 15 ) THEN
	
			Lt_WriteIndex	:= Lt_WriteIndex + 1;
			Step_SEQ		:= 35;	
						
		ELSIF ( Lt_WriteIndex <= 16 ) THEN
			
			Lt_ReadIndex	:= 0;
			Step_SEQ		:= 10;
		END_IF	
	
	999:
		xError	:= TRUE;
						
END_CASE

ReadPara(
	xExecute:= Lt_Execute_Read, 
	sNetId:=Lt_Read_Parameter_ISDU.Net_Id , 
	uiEthercatAddress:=Lt_Read_Parameter_ISDU.Ethercat_Address , 
	uiSlotNumber:=Lt_Read_Parameter_ISDU.Slot_Number , 
	usiPort:=Lt_Read_Parameter_ISDU.Port_Number , 
	uiIndex:=Lt_Read_Parameter_ISDU.Para_Index , 
	usiSubIndex:=Lt_Read_Parameter_ISDU.Para_SubIndex , 
	pData:=ADR(Lt_Read_Parameter_ISDU.Para_Data[0]) , 
	uiDataLength:=Lt_Read_Parameter_ISDU.Para_Length , 
	xWrite:=FALSE , 
	xIsString:=Lt_IsItString , 
	xDone=> , 
	xBusy=> , 
	xError=> , 
	udiErrorCode=> , 
	eErrorDescription=> , 
	udiReadDataLength=> );
	
	WritePara(
	xExecute:=Lt_Execute_Write , 
	sNetId:=Lt_Write_Parameter_ISDU.Net_Id , 
	uiEthercatAddress:=Lt_Write_Parameter_ISDU.Ethercat_Address , 
	uiSlotNumber:=Lt_Write_Parameter_ISDU.Slot_Number , 
	usiPort:=Lt_Write_Parameter_ISDU.Port_Number , 
	uiIndex:=Lt_Write_Parameter_ISDU.Para_Index , 
	usiSubIndex:=Lt_Write_Parameter_ISDU.Para_SubIndex , 
	pData:=ADR(Lt_Write_Parameter_ISDU.Para_Data[0]) , 
	uiDataLength:=Lt_Write_Parameter_ISDU.Para_Length , 
	xWrite:=TRUE , 
	xIsString:=FALSE , 
	xDone=> , 
	xBusy=> , 
	xError=> , 
	udiErrorCode=> , 
	eErrorDescription=> , 
	udiReadDataLength=> );
	
	// Current Position Feedback Value | Read Parameter Logic------------------------------------------------------------

diCurrentPosition 				:=  Lt_ReadParaData[0].Value;
Lt_ReadParaData[0].Sub_index	:= 16#0;
Lt_ReadParaData[0].Index		:= 16#120;
Lt_ReadParaData[0].Length		:= 4;

// Current Speed Feedback Value | Read Parameter Logic---------------------------------------------------------------
diCurrentSpeed 					:=  Lt_ReadParaData[1].Value;
Lt_ReadParaData[1].Sub_index	:= 16#0;
Lt_ReadParaData[1].Index		:= 16#121;
Lt_ReadParaData[1].Length		:= 4;

// Current Force Feedback Value | Read Parameter Logic---------------------------------------------------------------
diCurrentForce 					:=  Lt_ReadParaData[2].Value;
Lt_ReadParaData[2].Sub_index	:= 16#0;
Lt_ReadParaData[2].Index		:= 16#122;
Lt_ReadParaData[2].Length		:= 4;

//Error Data Feedback Value | Read Parameter Logic------------------------------------------------------------------
aErrorCode[0]	:= (Lt_ErrorRawData[2]) + SHL(TO_WORD(Lt_ErrorRawData[1]),8);
aErrorCode[1]	:= (Lt_ErrorRawData[5]) + SHL(TO_WORD(Lt_ErrorRawData[4]),8);
aErrorCode[2]	:= (Lt_ErrorRawData[8]) + SHL(TO_WORD(Lt_ErrorRawData[7]),8);
aErrorCode[3]	:= (Lt_ErrorRawData[11]) + SHL(TO_WORD(Lt_ErrorRawData[10]),8);
aErrorCode[4]	:= (Lt_ErrorRawData[14]) + SHL(TO_WORD(Lt_ErrorRawData[13]),8);
aErrorCode[5]	:= (Lt_ErrorRawData[17]) + SHL(TO_WORD(Lt_ErrorRawData[16]),8);
aErrorCode[6]	:= (Lt_ErrorRawData[20]) + SHL(TO_WORD(Lt_ErrorRawData[19]),8);
aErrorCode[7]	:= (Lt_ErrorRawData[23]) + SHL(TO_WORD(Lt_ErrorRawData[22]),8);
aErrorCode[8]	:= (Lt_ErrorRawData[26]) + SHL(TO_WORD(Lt_ErrorRawData[25]),8);
aErrorCode[9]	:= (Lt_ErrorRawData[29]) + SHL(TO_WORD(Lt_ErrorRawData[28]),8);
aErrorCode[10]	:= (Lt_ErrorRawData[32]) + SHL(TO_WORD(Lt_ErrorRawData[31]),8);
aErrorCode[11]	:= (Lt_ErrorRawData[35]) + SHL(TO_WORD(Lt_ErrorRawData[34]),8);
aErrorCode[12]	:= (Lt_ErrorRawData[38]) + SHL(TO_WORD(Lt_ErrorRawData[37]),8);
aErrorCode[13]	:= (Lt_ErrorRawData[41]) + SHL(TO_WORD(Lt_ErrorRawData[40]),8);
aErrorCode[14]	:= (Lt_ErrorRawData[44]) + SHL(TO_WORD(Lt_ErrorRawData[43]),8);
aErrorCode[15]	:= (Lt_ErrorRawData[47]) + SHL(TO_WORD(Lt_ErrorRawData[46]),8);

Lt_ReadParaData[3].Sub_index	:= 16#0;
Lt_ReadParaData[3].Index		:= 16#25;
Lt_ReadParaData[3].Length		:= 48;

// Current Temprature Feedback Value | Read Parameter Logic---------------------------------------------------------
diDDTemprature 					:=  Lt_ReadParaData[4].Value;
Lt_ReadParaData[4].Sub_index	:= 16#0;
Lt_ReadParaData[4].Index		:= 16#123;
Lt_ReadParaData[4].Length		:= 2;

// Actual Drive Current Feedback Value | Read Parameter Logic-------------------------------------------------------
diDDCurrent 					:=  Lt_ReadParaData[5].Value;
Lt_ReadParaData[5].Sub_index	:= 16#0;
Lt_ReadParaData[5].Index		:= 16#124;
Lt_ReadParaData[5].Length		:= 4;

// Actual Drive Voltage Feedback Value | Read Parameter Logic-------------------------------------------------------
diDDVoltage 					:=  Lt_ReadParaData[6].Value;
Lt_ReadParaData[6].Sub_index	:= 16#0;
Lt_ReadParaData[6].Index		:= 16#125;
Lt_ReadParaData[6].Length		:= 4;

// Axis Total Cycle Feedback Value | Read Parameter Logic-----------------------------------------------------------
diDDCyclesTotal 				:=  Lt_ReadParaData[7].Value;
Lt_ReadParaData[7].Sub_index	:= 16#0;
Lt_ReadParaData[7].Index		:= 16#126;
Lt_ReadParaData[7].Length		:= 4;

// Axis Cycle Since Reset Feedback Value | Read Parameter Logic------------------------------------------------------
diDDCyclesSinceReset			:=  Lt_ReadParaData[8].Value;
Lt_ReadParaData[8].Sub_index	:= 16#0;
Lt_ReadParaData[8].Index		:= 16#127;
Lt_ReadParaData[8].Length		:= 4;

// Axis Mileages Feedback Value | Read Parameter Logic---------------------------------------------------------------
diDDMileageTotal				:=  Lt_ReadParaData[9].Value;
Lt_ReadParaData[9].Sub_index	:= 16#0;
Lt_ReadParaData[9].Index		:= 16#128;
Lt_ReadParaData[9].Length		:= 4;

// Axis Mileages Since Reset Feedback Value | Read Parameter Logic--------------------------------------------------
diDDMileagesSinceReset			:=  Lt_ReadParaData[10].Value;
Lt_ReadParaData[10].Sub_index	:= 16#0;
Lt_ReadParaData[10].Index	:= 16#129;
Lt_ReadParaData[10].Length		:= 4;

// Number of Storage Operation Feedback Value | Read Parameter Logic--------------------------------------------------
diNumOfStorageOperation			:= Lt_NumOfStorageOperation / 2;
Lt_NumOfStorageOperation		:= Lt_ReadParaData[11].Value;
Lt_ReadParaData[11].Sub_index	:= 16#0;
Lt_ReadParaData[11].Index	    := 16#10A;
Lt_ReadParaData[11].Length		:= 4;

END_FUNCTION_BLOCK

// POUs/SMS_Festo_Basic
 FUNCTION_BLOCK SMS_Festo_Basic
VAR_INPUT
	RefINPUTS: BYTE;					//Input Channel Mapping
	xEnable: BOOL; 						//True - Enable AOI function
	sNetId              : STRING;
	uiEthercatAddress   : UINT;          //Address of the slave device i.e. CPX-AP-I-EC-M12 Module
	uiSlotNumber        : UINT;          //Slot number where the IO Link master CPX-AP-I-4IOL-M12 module is connected
	usiPort             : USINT;          //Port of the CPX-AP-I-4IOL-M12 module where IO link device is connected
	xMoveIN: BOOL;						//TRUE - SMS moves inwards | FALSE - SMS Stops		
	xMoveIntermediate: BOOL;			//TRUE – SMS Moves to Intermediate Position | FALSE – SMS Stops
	xMoveOut: BOOL;						//TRUE - SMS moves outwards | FALSE - SMS Stops
	xQuitError: BOOL;					//TRUE - Reset Error Messages
	xPowerSMS: BOOL;					//TRUE - Enable power stage of SMS
	xUserInterfaceLock: BOOL;			//TRUE - lock user interface of SMS control unit
	bySpeedOut: BYTE := 1;				//Axix Move Speed Towards Out Direction 1 - 10% (default) | Limit 1 to 10
	bySpeedIN: BYTE:= 1;				//Axix Move Speed Towards IN Direction 1 - 10% (default) | Limit 1 to 10
	byForce: BYTE:= 1;					//Axix Move Force 1 - 10% (default) | Limit 1 to 10
	xReferenceDirection: BOOL;			//TRUE - Motor averted | FALSE - Motor side
	xExecuteReference: BOOL;			//TRUE – Start Homing
	diStartPressPosition: DINT:= 100;	//Defines Start Position of Stroke
	diIntermediatePosition: DINT:= 200;	//Defines Intermediate Position of Stroke
	diEndPosition: DINT:= 300;			//Defines End Position of Stroke
	xAutoStoreActive: BOOL;				//TRUE – Automatically stores the last downloaded parameters in the SMS.
	xStoreParameters: BOOL;				//TRUE – Manually stores the last downloaded parameters in the SMS.
END_VAR
VAR_OUTPUT
	RefOUTPUTS: BYTE;					//Output Channel Mapping
	xEnabled: BOOL;						//TRUE - AOI Function Enabled
	xWriteActive: BOOL;					//TRUE - Executing Parameter Write Function
	xWriteDone: BOOL;					//TRUE - Last Parameter Wrote Successful
	xReadActive: BOOL;					//TRUE - Parameter Read Function is Active
	xStateIn: BOOL;						//TRUE - SMS Axis Reached IN Position
	xStateIntermediate: BOOL;			//TRUE - SMS Axis Reached Intermediate Position
	xStateOut: BOOL;					//TRUE - SMS Axis Reached OUT Position
	xStateMove: BOOL;					//TRUE – SMS Axis at Moving Condition | FALSE – SMS Axis at Ideal Condition
	xError: BOOL;						//TRUE - SMS Module or AOI in Error State. Check Error Code
	uiLocalError: UINT;					//Function Block Local Error Code
	aErrorCode: ARRAY[0..15] OF WORD;	//SMS Error Code List
	diCurrentPosition: DINT;			//Axis Current Position Feedback
	diCurrentSpeed: DINT;				//Axis Current Speed Feedback
	diCurrentForce: DINT;				//Axis Current Force Feedback
END_VAR
VAR
	Lt_ReadParaData: ARRAY[0..19] OF UDT_ReadParameter;
	Lt_WriteParaData: ARRAY[0..19] OF UDT_WriteParameter;
	Lt_ErrorRawData: ARRAY [0..48] OF BYTE;
	Lt_RiseEdgePowerSMS: BOOL;
	Lt_FalingEdgePowerSMS: BOOL;
	Lt_RiseUserInterfaceLock: BOOL;
	Lt_FalingEdgeUserInterfaceLock: BOOL;
	Lt_RiseReferenceDirection: BOOL;
	Lt_FalingEdgeReferenceDirection: BOOL;
	Lt_RiseExecuteReference: BOOL;
	Lt_FalingEdgeExecuteReference: BOOL;
	Lt_RiseStoreParameters: BOOL;
	Lt_FalingEdgeStoreParameters: BOOL;
	Lt_RiseResetCounterMileage: BOOL;
	Lt_FalingEdgeResetCounterMileage: BOOL;
	Lt_RiseAutoStoreActive: BOOL;
	Lt_FalingEdgeAutoStoreActive: BOOL;
	Lt_RiseEnableFileHandling: BOOL;
	Lt_FalingEdgeEnableFileHandling: BOOL;
	Step_SEQ: INT;
	Lt_ReadIndex: INT;
	Lt_WriteIndex: INT;
	Lt_Read_Parameter_ISDU: UDT_ISDU_Command;
	Lt_Write_Parameter_ISDU: UDT_ISDU_Command;
	Lt_ForLength: INT;
	Lt_Execute_Read: BOOL;
	Lt_Execute_Write: BOOL; 
	Lt_StateDevice: BOOL;
	Lt_ScanCount: DINT;
	Lt_ScanCount02: DINT;
	Lt_ScanCount03: DINT;
	Lt_ScanCount001: DINT;
	Lt_DeviceState_RisingEdge: BOOL;
	Lt_RealConvert: aByte_as_real;
	Lt_ExecuteReference_RisingEdge: BOOL;
	Lt_ExecuteReference_Trigger: BOOL;
	Lt_ExecuteReference_Trigger01: BOOL;	
	Lt_IsItString: BOOL;
	Lt_Startposition: REAL;
	Lt_Intermediateposition: REAL;
	Lt_Endposition: REAL;
	Lt_ReCurrentPosition: REAL;
	LT_ParameterRewriteDelay: BOOL;
	Lt_ExecuteReference_Trigger02: BOOL;
	
	ReadPara: CPXAPI_IOLink_Parameter;
	WritePara: CPXAPI_IOLink_Parameter;
	Delay_Timmer: TON;
	Elapse_time: TIME;
END_VAR

(*
===============================================================================================================
Advice TO Released Library Revisions 
===============================================================================================================
SMS_Festo_Lib | Communication: Beckhoff EtherCat
---------------------------------------------------------------------------------------------------------------
Version                           Date of Release
V1.0                                07.01.2022
V1.1                                03.06.2022

---------------------------------------------------------------------------------------------------------------
Changes in Library:

V1.0 -  Release Version


V1.1 - Position variables datatype changed from Real to Dint.
       Autostorage parameter continuous count bug fixed.
       Number of storage parameter double count bug fixed. 
*)
// Enable Function Block Sequence Logic------------------------------------------------------------------------ 
IF xEnable THEN 				
	xEnabled					:= TRUE;
	
ELSE
	xEnabled					:= FALSE;
	xWriteActive				:= FALSE;	
	xWriteDone					:= FALSE;
	xReadActive					:= FALSE;
	Step_SEQ					:= 0;
	Lt_ReadParaData[0].Value	:= 0;
	Lt_ReadParaData[1].Value	:= 0;
	Lt_ReadParaData[2].Value	:= 0;
	Lt_ReadParaData[3].Value	:= 0;
	
	
END_IF

//Process Data Command Logic---------------------------------------------------------------------------------------
IF xEnabled THEN				
	
	IF xMoveIN THEN				// Move IN Position Command
		RefOUTPUTS.0	:= TRUE;
	ELSE
		RefOUTPUTS.0	:= FALSE;
	END_IF
	
	IF xMoveOut THEN			// Move OUT Position Command
		RefOUTPUTS.1	:= TRUE;
	ELSE
		RefOUTPUTS.1	:= FALSE;	
	END_IF
	
	IF xMoveIntermediate THEN	// Move Intermediat Position Command
		RefOUTPUTS.4	:= TRUE;
	ELSE
		RefOUTPUTS.4	:= FALSE;	
	END_IF
	
	IF xQuitError THEN			// Move Quite Error Command
		RefOUTPUTS.2	:= TRUE;
	ELSE
		RefOUTPUTS.2	:= FALSE;	
	END_IF
ELSE							// Clear Command When FB Not Enabled
	RefOUTPUTS.0	:= FALSE;	
	RefOUTPUTS.1	:= FALSE;	
	RefOUTPUTS.2	:= FALSE;
	RefOUTPUTS.4	:= FALSE;
END_IF


// Process Data Feedback Logic---------------------------------------------------------------------------------
IF xEnabled THEN				
	
	IF RefINPUTS.0 THEN				// IN Position Status
		xStateIn	:= TRUE;
	ELSE
		xStateIn	:= FALSE;
	END_IF
	
	IF RefINPUTS.1 THEN				// Out Position Status
		xStateOut	:= TRUE;
	ELSE
		xStateOut	:= FALSE;
	END_IF
	
	IF RefINPUTS.2 THEN				// Axis Moving Status
		xStateMove	:= TRUE;
	ELSE
		xStateMove	:= FALSE;
	END_IF
	
	IF RefINPUTS.3 THEN				// Device Healthy Status
		Lt_StateDevice	:= TRUE;
	ELSE
		Lt_StateDevice	:= FALSE;
	END_IF
	
	IF RefINPUTS.4 THEN				// Intermediat Position Status
		xStateIntermediate	:= TRUE;
	ELSE
		xStateIntermediate	:= FALSE;
	END_IF	
ELSE 								// Clear Status When FB is Not Enabled
	xStateIn			:= FALSE;
	xStateOut			:= FALSE;
	xStateMove			:= FALSE;
	xStateIntermediate	:= FALSE;
	Lt_StateDevice		:= FALSE;
END_IF

// Device Error State Logic -----------------------------------------------------------------------------------
IF xEnabled AND xStateIn AND xStateOut AND NOT Lt_StateDevice THEN
	xError	:= TRUE;
ELSE
	xError	:= FALSE;
END_IF

// After Homing Parameters Re-Write Logic ---------------------------------------------------------------------
IF Lt_ExecuteReference_Trigger01	AND NOT xStateMove THEN
	Lt_ExecuteReference_Trigger02:= TRUE;
	
	IF LT_ParameterRewriteDelay THEN
		Lt_WriteParaData[0].PreviousValue	:= 0;
		Lt_WriteParaData[1].PreviousValue	:= 0;
		Lt_WriteParaData[2].PreviousValue	:= 0;
		Lt_WriteParaData[3].PreviousValue	:= 0;
		Lt_WriteParaData[4].PreviousValue	:= 0;
		Lt_WriteParaData[5].PreviousValue	:= 0;
		Lt_WriteParaData[7].PreviousValue	:= 0;
		Lt_WriteParaData[8].PreviousValue	:= 0;
		Lt_WriteParaData[9].PreviousValue	:= 0;
		Lt_WriteParaData[10].PreviousValue	:= 0;
		Lt_WriteParaData[11].PreviousValue	:= 0;
		Lt_ExecuteReference_Trigger01		:= FALSE;
		Lt_ExecuteReference_Trigger02       := FALSE;
		
	END_IF
ELSE
		Lt_ExecuteReference_Trigger02       := FALSE;
		
END_IF

// After Homing Parameter Rewrite Delay
Delay_Timmer(IN:= Lt_ExecuteReference_Trigger02, PT:=T#6S , Q=> LT_ParameterRewriteDelay, ET=> Elapse_time );

//Setpoint Limit Error-----------------------------------------------------------------------------------------
IF (bySpeedIN < 1 ) OR (bySpeedIN > 10 ) THEN 
	uiLocalError := 1001;
	xError		 := TRUE;

ELSIF (bySpeedOut < 1 ) OR (bySpeedOut > 10 ) THEN
	uiLocalError := 1002;
	xError		 := TRUE;
ELSIF (bySpeedIN < 1 ) OR (bySpeedIN > 10 ) THEN
	uiLocalError := 1003;
	xError		 := TRUE;
END_IF

//Device Status Rising Edge Logic--------------------------------------------------------------------------------
IF Lt_StateDevice AND NOT Lt_DeviceState_RisingEdge THEN
	Lt_DeviceState_RisingEdge	:= TRUE;
	xError						:= FALSE;
ELSIF NOT Lt_StateDevice THEN
	Lt_DeviceState_RisingEdge	:= FALSE;
END_IF

//Execute Ref Rising Edge Logic--------------------------------------------------------------------------------
IF xExecuteReference AND NOT Lt_ExecuteReference_RisingEdge THEN
	Lt_ExecuteReference_RisingEdge	:= TRUE;
	Lt_ExecuteReference_Trigger		:= TRUE;
	xError							:= FALSE;
ELSIF NOT xExecuteReference THEN
	Lt_ExecuteReference_RisingEdge	:= FALSE;
END_IF

// Quite Error Logic ------------------------------------------------------------------------------------------
IF xQuitError AND xEnabled THEN
	Step_SEQ			:= 0;
	xWriteActive		:= FALSE;
	xWriteDone			:= FALSE;
	xReadActive			:= FALSE;
	xError				:= FALSE;
	uiLocalError		:= 0;	
	
	// Clear Error Data Raw Array
		
	Lt_ErrorRawData[0] 		:= 0; Lt_ErrorRawData[1] 	:= 0; Lt_ErrorRawData[2] 	:= 0; Lt_ErrorRawData[3] 	:= 0;
	Lt_ErrorRawData[4] 		:= 0; Lt_ErrorRawData[5] 	:= 0; Lt_ErrorRawData[6] 	:= 0; Lt_ErrorRawData[7] 	:= 0;
	Lt_ErrorRawData[8] 		:= 0; Lt_ErrorRawData[9] 	:= 0; Lt_ErrorRawData[10] 	:= 0; Lt_ErrorRawData[11] 	:= 0;
	Lt_ErrorRawData[12] 	:= 0; Lt_ErrorRawData[13] 	:= 0; Lt_ErrorRawData[14] 	:= 0; Lt_ErrorRawData[15] 	:= 0;
	Lt_ErrorRawData[16] 	:= 0; Lt_ErrorRawData[17] 	:= 0; Lt_ErrorRawData[18] 	:= 0; Lt_ErrorRawData[19] 	:= 0;
	Lt_ErrorRawData[20] 	:= 0; Lt_ErrorRawData[21] 	:= 0; Lt_ErrorRawData[22] 	:= 0; Lt_ErrorRawData[23] 	:= 0;
	Lt_ErrorRawData[24] 	:= 0; Lt_ErrorRawData[25] 	:= 0; Lt_ErrorRawData[26] 	:= 0; Lt_ErrorRawData[27] 	:= 0;
	Lt_ErrorRawData[28] 	:= 0; Lt_ErrorRawData[29] 	:= 0; Lt_ErrorRawData[30] 	:= 0; Lt_ErrorRawData[31] 	:= 0;
	Lt_ErrorRawData[32] 	:= 0; Lt_ErrorRawData[33] 	:= 0; Lt_ErrorRawData[34] 	:= 0; Lt_ErrorRawData[35] 	:= 0;
	Lt_ErrorRawData[36] 	:= 0; Lt_ErrorRawData[37] 	:= 0; Lt_ErrorRawData[38] 	:= 0; Lt_ErrorRawData[39] 	:= 0;
	Lt_ErrorRawData[40] 	:= 0; Lt_ErrorRawData[41] 	:= 0; Lt_ErrorRawData[42] 	:= 0; Lt_ErrorRawData[43] 	:= 0;
	Lt_ErrorRawData[44] 	:= 0; Lt_ErrorRawData[45] 	:= 0; Lt_ErrorRawData[46] 	:= 0; Lt_ErrorRawData[47] 	:= 0;
	Lt_ErrorRawData[48] 	:= 0;	
	
END_IF

//Power Stage Enable & Disable Command Write Input Parameter Logic----------------------------------------------
IF xPowerSMS AND NOT Lt_RiseEdgePowerSMS THEN
	Lt_WriteParaData[0].NeedAction	:= TRUE;
	Lt_RiseEdgePowerSMS				:=	TRUE;
	Lt_FalingEdgePowerSMS			:=	FALSE;
	Lt_WriteParaData[0].Value		:= 16#0CC;
	
ELSIF NOT xPowerSMS	AND NOT Lt_FalingEdgePowerSMS THEN
	Lt_WriteParaData[0].NeedAction	:= TRUE;
	Lt_RiseEdgePowerSMS				:=	FALSE;
	Lt_FalingEdgePowerSMS			:=	TRUE;
	Lt_WriteParaData[0].Value		:= 16#0CB;
END_IF;


Lt_WriteParaData[0].Index		:= 2;
Lt_WriteParaData[0].Length			:= 1;
Lt_WriteParaData[0].Sub_index		:= 0;

//User Interface Lock Command Write Parameter Logic------------------------------------------------------------- 
IF xUserInterfaceLock AND NOT Lt_RiseUserInterfaceLock THEN
	Lt_WriteParaData[1].NeedAction	:= TRUE;
	Lt_RiseUserInterfaceLock 		:= TRUE;
	Lt_FalingEdgeUserInterfaceLock	:= FALSE;
	Lt_WriteParaData[1].Value		:= 1;
	
ELSIF NOT xUserInterfaceLock	AND NOT Lt_FalingEdgeUserInterfaceLock THEN
	Lt_WriteParaData[1].NeedAction	:= TRUE;
	Lt_RiseUserInterfaceLock		:= FALSE;
	Lt_FalingEdgeUserInterfaceLock	:= TRUE;
	Lt_WriteParaData[1].Value		:= 0;
END_IF;


Lt_WriteParaData[1].Index		:= 16#000C;
Lt_WriteParaData[1].Length			:= 1;
Lt_WriteParaData[1].Sub_index		:= 16#4;

//Speed Out % Command Write Parameter Logic--------------------------------------------------------------------- 
IF Lt_WriteParaData[2].Value <> Lt_WriteParaData[2].PreviousValue THEN 
	Lt_WriteParaData[2].NeedAction	:= TRUE;	
ELSE
	Lt_WriteParaData[2].NeedAction	:= FALSE;
	
END_IF

Lt_WriteParaData[2].Value			:= bySpeedOut;
Lt_WriteParaData[2].Sub_index		:= 16#0;
Lt_WriteParaData[2].Index		:= 16#101;
Lt_WriteParaData[2].Length			:= 1;


//Speed IN % Command Write Parameter Logic---------------------------------------------------------------------- 
IF Lt_WriteParaData[3].Value <> Lt_WriteParaData[3].PreviousValue THEN 
	Lt_WriteParaData[3].NeedAction	:= TRUE;	
ELSE
	Lt_WriteParaData[3].NeedAction	:= FALSE;
END_IF

Lt_WriteParaData[3].Value			:= bySpeedIN;
Lt_WriteParaData[3].Sub_index		:= 16#0;
Lt_WriteParaData[3].Index		:= 16#100;
Lt_WriteParaData[3].Length			:= 1;


//Force % Command Write Parameter Logic------------------------------------------------------------------------ 
IF Lt_WriteParaData[4].Value <> Lt_WriteParaData[4].PreviousValue THEN 
	Lt_WriteParaData[4].NeedAction	:= TRUE;	
ELSE
	Lt_WriteParaData[4].NeedAction	:= FALSE;
END_IF

Lt_WriteParaData[4].Value			:= byForce;
Lt_WriteParaData[4].Sub_index		:= 16#0;
Lt_WriteParaData[4].Index		:= 16#102;
Lt_WriteParaData[4].Length			:= 1;


//Referance Direction Command Write Parameter Logic----------------------------------------------------------- 
IF xReferenceDirection AND NOT Lt_RiseReferenceDirection THEN
	Lt_WriteParaData[5].NeedAction	:= TRUE;
	Lt_RiseReferenceDirection 		:= TRUE;
	Lt_FalingEdgeReferenceDirection	:= FALSE;
	Lt_WriteParaData[5].Value		:= 1;
	
ELSIF NOT xReferenceDirection	AND NOT Lt_FalingEdgeReferenceDirection THEN
	Lt_WriteParaData[5].NeedAction	:= TRUE;
	Lt_RiseReferenceDirection 		:= FALSE;
	Lt_FalingEdgeReferenceDirection	:= TRUE;
	Lt_WriteParaData[5].Value		:= 0;
END_IF;


Lt_WriteParaData[5].Index		:= 16#103;
Lt_WriteParaData[5].Length			:= 1;
Lt_WriteParaData[5].Sub_index		:= 16#0;

//Execute Referance Command | Write Parameter Logic------------------------------------------------------------ 
IF Lt_ExecuteReference_Trigger  THEN
	Lt_WriteParaData[6].NeedAction	:= TRUE;
	Lt_WriteParaData[6].Value		:= 1;
	Lt_ExecuteReference_Trigger		:= FALSE;
	Lt_ExecuteReference_Trigger01	:= TRUE;
		
ELSIF NOT xExecuteReference	 THEN
	Lt_WriteParaData[6].Value		:= 0;
END_IF;


Lt_WriteParaData[6].Index		:= 16#104;
Lt_WriteParaData[6].Length			:= 1;
Lt_WriteParaData[6].Sub_index		:= 16#0;

//Start Press Position Command | Write Parameter Logic---------------------------------------------------------- 
IF Lt_WriteParaData[9].Value <> Lt_WriteParaData[9].PreviousValue THEN 
	Lt_WriteParaData[9].NeedAction	:= TRUE;	
ELSE
	Lt_WriteParaData[9].NeedAction	:= FALSE;
END_IF


Lt_WriteParaData[9].REAL_Value		:= TO_REAL(diStartPressPosition);
Lt_WriteParaData[9].Value			:= diStartPressPosition;
Lt_WriteParaData[9].Sub_index		:= 16#0;
Lt_WriteParaData[9].Index		:= 16#105;
Lt_WriteParaData[9].Length			:= 4;


//End Position Command | Write Parameter Logic------------------------------------------------------------------- 
IF Lt_WriteParaData[7].Value <> Lt_WriteParaData[7].PreviousValue THEN 
	Lt_WriteParaData[7].NeedAction	:= TRUE;	
ELSE
	Lt_WriteParaData[7].NeedAction	:= FALSE;
END_IF

Lt_WriteParaData[7].REAL_Value		:= TO_REAL(diEndPosition);
Lt_WriteParaData[7].Value			:= diEndPosition;
Lt_WriteParaData[7].Sub_index		:= 16#0;
Lt_WriteParaData[7].Index		:= 16#106;
Lt_WriteParaData[7].Length			:= 4;


//Store Parameters Command | Write Parameter Logic--------------------------------------------------------------- 
IF xStoreParameters AND NOT Lt_RiseStoreParameters AND xEnabled THEN
	Lt_WriteParaData[10].NeedAction	:= TRUE;
	Lt_RiseStoreParameters 			:= TRUE;
	Lt_FalingEdgeStoreParameters	:= FALSE;
	Lt_WriteParaData[10].Value		:= 1;
	
ELSIF NOT xStoreParameters	AND NOT Lt_FalingEdgeStoreParameters AND xEnabled THEN
	Lt_WriteParaData[10].NeedAction	:= TRUE;
	Lt_RiseStoreParameters  		:= FALSE;
	Lt_FalingEdgeStoreParameters	:= TRUE;
	Lt_WriteParaData[10].Value		:= 0;
END_IF;


Lt_WriteParaData[10].Index		:= 16#10B;
Lt_WriteParaData[10].Length			:= 1;
Lt_WriteParaData[10].Sub_index		:= 16#0;

//Intermediate Position Command | Write Parameter Logic ------------------------------------------------------------
IF Lt_WriteParaData[8].Value <> Lt_WriteParaData[8].PreviousValue THEN 
	Lt_WriteParaData[8].NeedAction	:= TRUE;	
ELSE
	Lt_WriteParaData[8].NeedAction	:= FALSE;
END_IF

Lt_WriteParaData[8].REAL_Value		:= TO_REAL(diIntermediatePosition);
Lt_WriteParaData[8].Value			:= diIntermediatePosition;
Lt_WriteParaData[8].Sub_index		:= 16#0;
Lt_WriteParaData[8].Index		:= 16#108;
Lt_WriteParaData[8].Length			:= 4;


//Auto Store Parameters Command | Write Parameter Logic------------------------------------------------------------- 
IF xAutoStoreActive AND NOT Lt_RiseAutoStoreActive  THEN
	Lt_WriteParaData[11].NeedAction	:= TRUE;
	Lt_RiseAutoStoreActive 			:= TRUE;
	Lt_FalingEdgeAutoStoreActive	:= FALSE;
	Lt_WriteParaData[11].Value		:= 1;
	
ELSIF NOT xAutoStoreActive	AND NOT Lt_FalingEdgeAutoStoreActive  THEN
	Lt_WriteParaData[11].NeedAction	:= TRUE;
	Lt_RiseAutoStoreActive  		:= FALSE;
	Lt_FalingEdgeAutoStoreActive	:= TRUE;
	Lt_WriteParaData[11].Value		:= 0;
END_IF;


Lt_WriteParaData[11].Index		:= 16#109;
Lt_WriteParaData[11].Length			:= 1;
Lt_WriteParaData[11].Sub_index		:= 16#0;

//Read & Write Control Sequence Logic-------------------------------------------------------------------------------
CASE Step_SEQ OF 					
	0:	// Enable Read & Write Logic
		IF xEnabled THEN 
			Lt_ReadIndex	:= 0;
			Lt_WriteIndex	:= 0;
			Step_SEQ		:= 10;
		ELSE
			Step_SEQ		:= 0;
		END_IF
	10:	// Read Data Parameter Input Logic 
		Lt_Read_Parameter_ISDU.Net_Id	        :=	sNetId ;
		Lt_Read_Parameter_ISDU.Ethercat_Address	:=	uiEthercatAddress ;
		Lt_Read_Parameter_ISDU.Slot_Number	    :=	uiSlotNumber ;
		Lt_Read_Parameter_ISDU.Port_Number		:=	usiPort;
		Lt_Read_Parameter_ISDU.Para_Index		:=	Lt_ReadParaData[Lt_ReadIndex].Index;
		Lt_Read_Parameter_ISDU.Para_SubIndex	:=	Lt_ReadParaData[Lt_ReadIndex].Sub_index;
		Lt_Read_Parameter_ISDU.Para_Length		:=	Lt_ReadParaData[Lt_ReadIndex].Length;
		Lt_Read_Parameter_ISDU.Para_Data[0]		:=	0;
		Lt_Read_Parameter_ISDU.Para_Data[1]		:=	0;
		Lt_Read_Parameter_ISDU.Para_Data[2]		:=	0;
		Lt_Read_Parameter_ISDU.Para_Data[3]		:=	0;
		
		IF (Lt_ReadIndex = 3)	THEN	// Is It String Command Mapping for Read Instruction 
			Lt_IsItString	:= TRUE;
			ELSE 
			Lt_IsItString	:= FALSE;
		END_IF
		
		xReadActive						:= TRUE;
		xWriteActive					:= FALSE;
		Step_SEQ						:= 20;
		
	20:	// Read Command Enable Logic 
		
			Lt_Execute_Read		:=	TRUE;	 
		 	Step_SEQ			:= 21;
			
	21: // Read Feedback Data Manipulation
		IF ReadPara.xDone	THEN
			
			IF Lt_ReadIndex <> 3 THEN
				Lt_ForLength	:= 0;
				IF 	(Lt_ReadParaData[Lt_ReadIndex].Length = 4) THEN
					Lt_ReadParaData[Lt_ReadIndex].Value	:= TO_DINT(Lt_Read_Parameter_ISDU.Para_Data[0]) + SHL(TO_DINT(Lt_Read_Parameter_ISDU.Para_Data[1]),8)	+ SHL(TO_DINT(Lt_Read_Parameter_ISDU.Para_Data[2]),16) 
														+ SHL(TO_DINT(Lt_Read_Parameter_ISDU.Para_Data[3]),24);
														
				ELSIF (Lt_ReadParaData[Lt_ReadIndex].Length = 2) THEN
					Lt_ReadParaData[Lt_ReadIndex].Value	:= TO_DINT(Lt_Read_Parameter_ISDU.Para_Data[0]) + SHL(TO_DINT(Lt_Read_Parameter_ISDU.Para_Data[1]),8);
			
				ELSIF (Lt_ReadParaData[Lt_ReadIndex].Length = 1) THEN
					Lt_ReadParaData[Lt_ReadIndex].Value	:= TO_DINT(Lt_Read_Parameter_ISDU.Para_Data[0]);
				END_IF;
					
			ELSE
			
				Lt_ErrorRawData[0] 		:= ReadPara.pData[0];	 Lt_ErrorRawData[1] := ReadPara.pData[1]; 	Lt_ErrorRawData[2] 	:= ReadPara.pData[2]; Lt_ErrorRawData[3] 	:= ReadPara.pData[3];
				Lt_ErrorRawData[4] 		:= ReadPara.pData[4]; 	Lt_ErrorRawData[5] 	:= ReadPara.pData[5];	Lt_ErrorRawData[6] 	:= ReadPara.pData[6]; Lt_ErrorRawData[7] 	:= ReadPara.pData[7];
				Lt_ErrorRawData[8] 		:= ReadPara.pData[8]; 	Lt_ErrorRawData[9] 	:= ReadPara.pData[9]; 	Lt_ErrorRawData[10] := ReadPara.pData[10]; Lt_ErrorRawData[11] 	:= ReadPara.pData[11];
				Lt_ErrorRawData[12] 	:= ReadPara.pData[12]; Lt_ErrorRawData[13] 	:= ReadPara.pData[13]; Lt_ErrorRawData[14] 	:= ReadPara.pData[14]; Lt_ErrorRawData[15] 	:= ReadPara.pData[15];
				Lt_ErrorRawData[16] 	:= ReadPara.pData[16]; Lt_ErrorRawData[17] 	:= ReadPara.pData[17]; Lt_ErrorRawData[18] 	:= ReadPara.pData[18]; Lt_ErrorRawData[19] 	:= ReadPara.pData[19];
				Lt_ErrorRawData[20] 	:= ReadPara.pData[20]; Lt_ErrorRawData[21] 	:= ReadPara.pData[21]; Lt_ErrorRawData[22] 	:= ReadPara.pData[22]; Lt_ErrorRawData[23] 	:= ReadPara.pData[23];
				Lt_ErrorRawData[24] 	:= ReadPara.pData[24]; Lt_ErrorRawData[25] 	:= ReadPara.pData[25]; Lt_ErrorRawData[26] 	:= ReadPara.pData[26]; Lt_ErrorRawData[27] 	:= ReadPara.pData[27];
				Lt_ErrorRawData[28] 	:= ReadPara.pData[28]; Lt_ErrorRawData[29] 	:= ReadPara.pData[29]; Lt_ErrorRawData[30] 	:= ReadPara.pData[30]; Lt_ErrorRawData[31] 	:= ReadPara.pData[31];
				Lt_ErrorRawData[32] 	:= ReadPara.pData[32]; Lt_ErrorRawData[33] 	:= ReadPara.pData[33]; Lt_ErrorRawData[34] 	:= ReadPara.pData[34]; Lt_ErrorRawData[35] 	:= ReadPara.pData[35];
				Lt_ErrorRawData[36] 	:= ReadPara.pData[36]; Lt_ErrorRawData[37] 	:= ReadPara.pData[37]; Lt_ErrorRawData[38] 	:= ReadPara.pData[38]; Lt_ErrorRawData[39] 	:= ReadPara.pData[39];
				Lt_ErrorRawData[40] 	:= ReadPara.pData[40]; Lt_ErrorRawData[41] 	:= ReadPara.pData[41]; Lt_ErrorRawData[42] 	:= ReadPara.pData[42]; Lt_ErrorRawData[43] 	:= ReadPara.pData[43];
				Lt_ErrorRawData[44] 	:= ReadPara.pData[44]; Lt_ErrorRawData[45] 	:= ReadPara.pData[45]; Lt_ErrorRawData[46] 	:= ReadPara.pData[46]; Lt_ErrorRawData[47] 	:= ReadPara.pData[47];
				Lt_ErrorRawData[48] 	:= ReadPara.pData[48];
			
			END_IF
			
			Lt_ScanCount03	:= Lt_ScanCount03 + 1;
			IF Lt_ScanCount03 > 2 THEN 
			Lt_Execute_Read					:= FALSE;
			Step_SEQ						:= 30;
			Lt_ScanCount03					:= 0;
			END_IF
			
		ELSIF	ReadPara.xError	THEN 
			
			uiLocalError					:= 1004;
			Lt_Execute_Read					:= FALSE;
			Step_SEQ						:= 999;
			
		END_IF
	30:	// Read Parameter List Index & Move Sequence to Write Function Logic
		IF ( Lt_ReadIndex <= 3 ) THEN
			
			Lt_ReadIndex 	:= Lt_ReadIndex + 1;
			Step_SEQ		:= 10;
		END_IF 
		
		IF  Lt_ReadIndex >= 4  THEN
			
			Lt_WriteIndex	:= 0;
			Step_SEQ		:= 35;
			
		END_IF
		
	35:	// Reset The Wrie ISDU Parameters Data
			Lt_Write_Parameter_ISDU.Para_Data[0]	:= 0;	
			Lt_Write_Parameter_ISDU.Para_Data[1]	:= 0;
			Lt_Write_Parameter_ISDU.Para_Data[2]	:= 0;
			Lt_Write_Parameter_ISDU.Para_Data[3]	:= 0;	
			Step_SEQ								:= 40;
			
	40:	// Write Data Parameter Input Logic 
		Lt_Write_Parameter_ISDU.Net_Id	:=	sNetId;
		Lt_Write_Parameter_ISDU.Ethercat_Address	:=	uiEthercatAddress;
		Lt_Write_Parameter_ISDU.Slot_Number	:=	uiSlotNumber;
		Lt_Write_Parameter_ISDU.Port_Number	:=	usiPort;
		Lt_Write_Parameter_ISDU.Para_Index	:=	Lt_WriteParaData[Lt_WriteIndex].Index;
		Lt_Write_Parameter_ISDU.Para_SubIndex	:=	Lt_WriteParaData[Lt_WriteIndex].Sub_index;
		Lt_Write_Parameter_ISDU.Para_Length		:=	Lt_WriteParaData[Lt_WriteIndex].Length;
		
		IF Lt_Write_Parameter_ISDU.Para_Length = 4 THEN
			
			Lt_RealConvert.rRealValue				:= Lt_WriteParaData[Lt_WriteIndex].REAL_Value;
			Lt_Write_Parameter_ISDU.Para_Data[0]	:= Lt_RealConvert.abyte[0];	
			Lt_Write_Parameter_ISDU.Para_Data[1]	:= Lt_RealConvert.abyte[1];
			Lt_Write_Parameter_ISDU.Para_Data[2]	:= Lt_RealConvert.abyte[2];
			Lt_Write_Parameter_ISDU.Para_Data[3]	:= Lt_RealConvert.abyte[3];	
		
		ELSIF Lt_Write_Parameter_ISDU.Para_Length = 2 THEN
			Lt_Write_Parameter_ISDU.Para_Data[0]	:=	TO_BYTE(Lt_WriteParaData[Lt_WriteIndex].Value);
			Lt_Write_Parameter_ISDU.Para_Data[1]	:=	TO_BYTE(SHR(Lt_WriteParaData[Lt_WriteIndex].Value,8));
		
		ELSIF Lt_Write_Parameter_ISDU.Para_Length = 1 THEN
			Lt_Write_Parameter_ISDU.Para_Data[0]	:=	TO_BYTE(Lt_WriteParaData[Lt_WriteIndex].Value);
		END_IF
		
		Lt_ScanCount	:= Lt_ScanCount + 1;
		
		IF 	Lt_ScanCount >= 2 THEN
		xReadActive						:= FALSE;
		//xWriteActive					:= TRUE;
		Lt_ScanCount					:= 0;	
		Step_SEQ						:= 50;
		END_IF
	
	50:	// Write Command Enable Logic 
		IF Lt_WriteIndex <> 7 THEN
            IF Lt_WriteParaData[Lt_WriteIndex].NeedAction THEN
                Lt_Execute_Write := TRUE;
                xWriteDone := FALSE;
				xReadActive	:= FALSE;
		        xWriteActive:= TRUE;
                Step_SEQ := 51;
            ELSE
                Step_SEQ := 60;
            END_IF;
        ELSE
            IF NOT Lt_ExecuteReference_Trigger01 THEN
                IF Lt_WriteParaData[Lt_WriteIndex].NeedAction THEN
                    Lt_Execute_Write := TRUE;
                    xWriteDone := FALSE;
					xReadActive	:= FALSE;
		            xWriteActive:= TRUE;
                    Step_SEQ := 51;
                ELSE
                    Step_SEQ := 60;
                END_IF;
            END_IF;
        END_IF;
		
	51:	// Write Data Manipulation
		IF WritePara.xDone THEN
			Lt_WriteParaData[Lt_WriteIndex].NeedAction		:= FALSE;
			Lt_WriteParaData[Lt_WriteIndex].PreviousValue	:= Lt_WriteParaData[Lt_WriteIndex].Value;
			Lt_Execute_Write								:= FALSE;
			xWriteDone										:= TRUE;
			xWriteActive									:= FALSE;
			Step_SEQ										:= 60;	 
		ELSIF WritePara.xError	THEN
			uiLocalError		:= 1005;
			Lt_Execute_Write	:= FALSE;
			Step_SEQ			:= 999;
		 END_IF
	
	60:	// Write Parameter List Index & Move Sequence to Read Function Logic
		IF ( Lt_WriteIndex <= 11 ) THEN
	
			Lt_WriteIndex	:= Lt_WriteIndex + 1;
			Step_SEQ		:= 35;	
						
		ELSIF ( Lt_WriteIndex >= 12 ) THEN
			
			Lt_ReadIndex	:= 0;
			Step_SEQ		:= 10;
		END_IF	
	
	999:
		xError	:= TRUE;
						
END_CASE

ReadPara(
	xExecute:= Lt_Execute_Read, 
	sNetId:=Lt_Read_Parameter_ISDU.Net_Id , 
	uiEthercatAddress:=Lt_Read_Parameter_ISDU.Ethercat_Address , 
	uiSlotNumber:=Lt_Read_Parameter_ISDU.Slot_Number , 
	usiPort:=Lt_Read_Parameter_ISDU.Port_Number , 
	uiIndex:=Lt_Read_Parameter_ISDU.Para_Index , 
	usiSubIndex:=Lt_Read_Parameter_ISDU.Para_SubIndex , 
	pData:=ADR(Lt_Read_Parameter_ISDU.Para_Data[0]) , 
	uiDataLength:=Lt_Read_Parameter_ISDU.Para_Length , 
	xWrite:=FALSE , 
	xIsString:=Lt_IsItString , 
	xDone=> , 
	xBusy=> , 
	xError=> , 
	udiErrorCode=> , 
	eErrorDescription=> , 
	udiReadDataLength=> );
	
	WritePara(
	xExecute:=Lt_Execute_Write , 
	sNetId:=Lt_Write_Parameter_ISDU.Net_Id , 
	uiEthercatAddress:=Lt_Write_Parameter_ISDU.Ethercat_Address , 
	uiSlotNumber:=Lt_Write_Parameter_ISDU.Slot_Number , 
	usiPort:=Lt_Write_Parameter_ISDU.Port_Number , 
	uiIndex:=Lt_Write_Parameter_ISDU.Para_Index , 
	usiSubIndex:=Lt_Write_Parameter_ISDU.Para_SubIndex , 
	pData:=ADR(Lt_Write_Parameter_ISDU.Para_Data[0]) , 
	uiDataLength:=Lt_Write_Parameter_ISDU.Para_Length , 
	xWrite:=TRUE , 
	xIsString:=FALSE , 
	xDone=> , 
	xBusy=> , 
	xError=> , 
	udiErrorCode=> , 
	eErrorDescription=> , 
	udiReadDataLength=> );
				 
				 
// Current Position Feedback Value | Read Parameter Logic------------------------------------------------------------
diCurrentPosition 				:=  Lt_ReadParaData[0].Value;
Lt_ReadParaData[0].Sub_index	:= 16#0;
Lt_ReadParaData[0].Index		:= 16#120;
Lt_ReadParaData[0].Length		:= 4;

// Current Speed Feedback Value | Read Parameter Logic---------------------------------------------------------------
diCurrentSpeed 					:=  Lt_ReadParaData[1].Value;
Lt_ReadParaData[1].Sub_index	:= 16#0;
Lt_ReadParaData[1].Index		:= 16#121;
Lt_ReadParaData[1].Length		:= 4;

// Current Force Feedback Value | Read Parameter Logic---------------------------------------------------------------
diCurrentForce 					:=  Lt_ReadParaData[2].Value;
Lt_ReadParaData[2].Sub_index	:= 16#0;
Lt_ReadParaData[2].Index		:= 16#122;
Lt_ReadParaData[2].Length		:= 4;

//Error Data Feedback Value | Read Parameter Logic------------------------------------------------------------------
aErrorCode[0]	:= (Lt_ErrorRawData[2]) + SHL(TO_WORD(Lt_ErrorRawData[1]),8);
aErrorCode[1]	:= (Lt_ErrorRawData[5]) + SHL(TO_WORD(Lt_ErrorRawData[4]),8);
aErrorCode[2]	:= (Lt_ErrorRawData[8]) + SHL(TO_WORD(Lt_ErrorRawData[7]),8);
aErrorCode[3]	:= (Lt_ErrorRawData[11]) + SHL(TO_WORD(Lt_ErrorRawData[10]),8);
aErrorCode[4]	:= (Lt_ErrorRawData[14]) + SHL(TO_WORD(Lt_ErrorRawData[13]),8);
aErrorCode[5]	:= (Lt_ErrorRawData[17]) + SHL(TO_WORD(Lt_ErrorRawData[16]),8);
aErrorCode[6]	:= (Lt_ErrorRawData[20]) + SHL(TO_WORD(Lt_ErrorRawData[19]),8);
aErrorCode[7]	:= (Lt_ErrorRawData[23]) + SHL(TO_WORD(Lt_ErrorRawData[22]),8);
aErrorCode[8]	:= (Lt_ErrorRawData[26]) + SHL(TO_WORD(Lt_ErrorRawData[25]),8);
aErrorCode[9]	:= (Lt_ErrorRawData[29]) + SHL(TO_WORD(Lt_ErrorRawData[28]),8);
aErrorCode[10]	:= (Lt_ErrorRawData[32]) + SHL(TO_WORD(Lt_ErrorRawData[31]),8);
aErrorCode[11]	:= (Lt_ErrorRawData[35]) + SHL(TO_WORD(Lt_ErrorRawData[34]),8);
aErrorCode[12]	:= (Lt_ErrorRawData[38]) + SHL(TO_WORD(Lt_ErrorRawData[37]),8);
aErrorCode[13]	:= (Lt_ErrorRawData[41]) + SHL(TO_WORD(Lt_ErrorRawData[40]),8);
aErrorCode[14]	:= (Lt_ErrorRawData[44]) + SHL(TO_WORD(Lt_ErrorRawData[43]),8);
aErrorCode[15]	:= (Lt_ErrorRawData[47]) + SHL(TO_WORD(Lt_ErrorRawData[46]),8);

Lt_ReadParaData[3].Sub_index	:= 16#0;
Lt_ReadParaData[3].Index		:= 16#25;
Lt_ReadParaData[3].Length		:= 48;

END_FUNCTION_BLOCK

// POUs/SMS_Festo_Intermediate
 FUNCTION_BLOCK SMS_Festo_Intermediate
VAR_INPUT
	RefINPUTS: BYTE;					//Input Channel Mapping
	xEnable: BOOL; 						//True - Enable AOI function
	sNetId              : STRING;
	uiEthercatAddress   : UINT;          //Address of the slave device i.e. CPX-AP-I-EC-M12 Module
	uiSlotNumber        : UINT;          //Slot number where the IO Link master CPX-AP-I-4IOL-M12 module is connected
	usiPort             : USINT;          //Port of the CPX-AP-I-4IOL-M12 module where IO link device is connected
	xMoveIN: BOOL;						//TRUE - SMS moves inwards | FALSE - SMS Stops		
	xMoveIntermediate: BOOL;			//TRUE – SMS Moves to Intermediate Position | FALSE – SMS Stops
	xMoveOut: BOOL;						//TRUE - SMS moves outwards | FALSE - SMS Stops
	xQuitError: BOOL;					//TRUE - Reset Error Messages
	diIntermediatePosition: DINT:= 200;	//Defines Intermediate Position of Stroke
	bySpeedOut: BYTE := 1;				//Axix Move Speed Towards Out Direction 1 - 10% (default) | Limit 1 to 10
	bySpeedIN: BYTE:= 1;				//Axix Move Speed Towards IN Direction 1 - 10% (default) | Limit 1 to 10
	
	
	
END_VAR	
	
VAR_OUTPUT
	
	RefOUTPUTS: BYTE;					//Output Channel Mapping
	xEnabled: BOOL;						//TRUE - AOI Function Enabled
	xStateIn: BOOL;						//TRUE - SMS Axis Reached IN Position
	xStateIntermediate: BOOL;			//TRUE - SMS Axis Reached Intermediate Position
	xStateOut: BOOL;					//TRUE - SMS Axis Reached OUT Position
	xStateMove: BOOL;					//TRUE – SMS Axis at Moving Condition | FALSE – SMS Axis at Ideal Condition
	xError: BOOL;						//TRUE - SMS Module or AOI in Error State. Check Error Code
	diCurrentPosition: DINT;			//Axis Current Position Feedback
	xWriteDone: BOOL;					//TRUE - Last Parameter Wrote Successful
	
	
END_VAR

VAR
	Lt_ReadParaData: ARRAY[0..19] OF UDT_ReadParameter;
	Lt_WriteParaData: ARRAY[0..19] OF UDT_WriteParameter;
	Lt_ErrorRawData: ARRAY [0..48] OF BYTE;
	Lt_RiseEdgePowerSMS: BOOL;
	Lt_FalingEdgePowerSMS: BOOL;
	Lt_RiseUserInterfaceLock: BOOL;
	Lt_FalingEdgeUserInterfaceLock: BOOL;
	Lt_RiseReferenceDirection: BOOL;
	Lt_FalingEdgeReferenceDirection: BOOL;
	Lt_RiseExecuteReference: BOOL;
	Lt_FalingEdgeExecuteReference: BOOL;
	Lt_RiseStoreParameters: BOOL;
	Lt_FalingEdgeStoreParameters: BOOL;
	Lt_RiseResetCounterMileage: BOOL;
	Lt_FalingEdgeResetCounterMileage: BOOL;
	Lt_RiseAutoStoreActive: BOOL;
	Lt_FalingEdgeAutoStoreActive: BOOL;
	Lt_RiseEnableFileHandling: BOOL;
	Lt_FalingEdgeEnableFileHandling: BOOL;
	Step_SEQ: INT;
	Lt_ReadIndex: INT;
	Lt_WriteIndex: INT;
	Lt_Read_Parameter_ISDU: UDT_ISDU_Command;
	Lt_Write_Parameter_ISDU: UDT_ISDU_Command;
	Lt_ForLength: INT;
	Lt_Execute_Read: BOOL;
	Lt_Execute_Write: BOOL; 
	Lt_StateDevice: BOOL;
	Lt_ScanCount: DINT;
	Lt_ScanCount02: DINT;
	Lt_ScanCount03: DINT;
	Lt_ScanCount001: DINT;
	Lt_DeviceState_RisingEdge: BOOL;
	Lt_RealConvert: aByte_as_real;
		
	Lt_IsItString: BOOL;
	Lt_Startposition: REAL;
	Lt_Intermediateposition: REAL;
	Lt_Endposition: REAL;
	Lt_ReCurrentPosition: REAL;
	LT_ParameterRewriteDelay: BOOL;
	Lt_ExecuteReference_Trigger02: BOOL;
	
	ReadPara: CPXAPI_IOLink_Parameter;
	WritePara: CPXAPI_IOLink_Parameter;
	Delay_Timmer: TON;
	Elapse_time: TIME;
END_VAR

(*
===============================================================================================================
Advice TO Released Library Revisions 
===============================================================================================================
SMS_Festo_Lib | Communication: Beckhoff EtherCat
---------------------------------------------------------------------------------------------------------------
Version                           Date of Release
V1.0                                07.01.2022
V1.1                                03.06.2022

---------------------------------------------------------------------------------------------------------------
Changes in Library:

V1.0 -  Release Version


V1.1 - Release version SMS_Festo_Intermediate block. 
*)




// Enable Function Block Sequence Logic------------------------------------------------------------------------ 
IF xEnable THEN 				
	xEnabled					:= TRUE;
	
ELSE
	xEnabled					:= FALSE;
	xWriteDone					:= FALSE;
	Step_SEQ					:= 0;
END_IF

//Process Data Command Logic---------------------------------------------------------------------------------------
IF xEnabled THEN				
	
	IF xMoveIN THEN				// Move IN Position Command
		RefOUTPUTS.0	:= TRUE;
	ELSE
		RefOUTPUTS.0	:= FALSE;
	END_IF
	
	IF xMoveOut THEN			// Move OUT Position Command
		RefOUTPUTS.1	:= TRUE;
	ELSE
		RefOUTPUTS.1	:= FALSE;	
	END_IF
	
	IF xMoveIntermediate THEN	// Move Intermediat Position Command
		RefOUTPUTS.4	:= TRUE;
	ELSE
		RefOUTPUTS.4	:= FALSE;	
	END_IF
	
	IF xQuitError THEN			// Move Quite Error Command
		RefOUTPUTS.2	:= TRUE;
	ELSE
		RefOUTPUTS.2	:= FALSE;	
	END_IF
ELSE							// Clear Command When FB Not Enabled
	RefOUTPUTS.0	:= FALSE;	
	RefOUTPUTS.1	:= FALSE;	
	RefOUTPUTS.2	:= FALSE;
	RefOUTPUTS.4	:= FALSE;
END_IF


// Process Data Feedback Logic---------------------------------------------------------------------------------
IF xEnabled THEN				
	
	IF RefINPUTS.0 THEN				// IN Position Status
		xStateIn	:= TRUE;
	ELSE
		xStateIn	:= FALSE;
	END_IF
	
	IF RefINPUTS.1 THEN				// Out Position Status
		xStateOut	:= TRUE;
	ELSE
		xStateOut	:= FALSE;
	END_IF
	
	IF RefINPUTS.2 THEN				// Axis Moving Status
		xStateMove	:= TRUE;
	ELSE
		xStateMove	:= FALSE;
	END_IF
	
	IF RefINPUTS.3 THEN				// Device Healthy Status
		Lt_StateDevice	:= TRUE;
	ELSE
		Lt_StateDevice	:= FALSE;
	END_IF
	
	IF RefINPUTS.4 THEN				// Intermediat Position Status
		xStateIntermediate	:= TRUE;
	ELSE
		xStateIntermediate	:= FALSE;
	END_IF	
ELSE 								// Clear Status When FB is Not Enabled
	xStateIn			:= FALSE;
	xStateOut			:= FALSE;
	xStateMove			:= FALSE;
	xStateIntermediate	:= FALSE;
	Lt_StateDevice		:= FALSE;
END_IF

// Device Error State Logic -----------------------------------------------------------------------------------
IF xEnabled AND xStateIn AND xStateOut AND NOT Lt_StateDevice THEN
	xError	:= TRUE;
ELSE
	xError	:= FALSE;
END_IF



//Setpoint Limit Error-----------------------------------------------------------------------------------------
IF (bySpeedIN < 1 ) OR (bySpeedIN > 10 ) THEN 
	xError		 := TRUE;

ELSIF (bySpeedOut < 1 ) OR (bySpeedOut > 10 ) THEN
		xError		 := TRUE;
ELSIF (bySpeedIN < 1 ) OR (bySpeedIN > 10 ) THEN
		xError		 := TRUE;
END_IF

//Device Status Rising Edge Logic--------------------------------------------------------------------------------
IF Lt_StateDevice AND NOT Lt_DeviceState_RisingEdge THEN
	Lt_DeviceState_RisingEdge	:= TRUE;
	xError						:= FALSE;
ELSIF NOT Lt_StateDevice THEN
	Lt_DeviceState_RisingEdge	:= FALSE;
END_IF


// Quite Error Logic ------------------------------------------------------------------------------------------
IF xQuitError AND xEnabled THEN
	Step_SEQ			:= 0;
	xWriteDone			:= FALSE;
	xError				:= FALSE;
		
END_IF

//Intermediate Position Command | Write Parameter Logic ------------------------------------------------------------
IF Lt_WriteParaData[0].Value <> Lt_WriteParaData[0].PreviousValue THEN 
	Lt_WriteParaData[0].NeedAction	:= TRUE;	
ELSE
	Lt_WriteParaData[0].NeedAction	:= FALSE;
END_IF
Lt_WriteParaData[0].REAL_Value		:= TO_REAL(diIntermediatePosition);
Lt_WriteParaData[0].Value			:= diIntermediatePosition;
Lt_WriteParaData[0].Sub_index		:= 16#0;
Lt_WriteParaData[0].Index		:= 16#108;
Lt_WriteParaData[0].Length			:= 4;

//Speed IN % Command Write Parameter Logic---------------------------------------------------------------------- 
IF Lt_WriteParaData[1].Value <> Lt_WriteParaData[1].PreviousValue THEN 
	Lt_WriteParaData[1].NeedAction	:= TRUE;	
ELSE
	Lt_WriteParaData[1].NeedAction	:= FALSE;
END_IF

Lt_WriteParaData[1].Value			:= bySpeedIN;
Lt_WriteParaData[1].Sub_index		:= 16#0;
Lt_WriteParaData[1].Index		:= 16#100;
Lt_WriteParaData[1].Length			:= 1;

//Speed Out % Command Write Parameter Logic--------------------------------------------------------------------- 
IF Lt_WriteParaData[2].Value <> Lt_WriteParaData[2].PreviousValue THEN 
	Lt_WriteParaData[2].NeedAction	:= TRUE;	
ELSE
	Lt_WriteParaData[2].NeedAction	:= FALSE;
	
END_IF

Lt_WriteParaData[2].Value			:= bySpeedOut;
Lt_WriteParaData[2].Sub_index		:= 16#0;
Lt_WriteParaData[2].Index		:= 16#101;
Lt_WriteParaData[2].Length			:= 1;



//Read & Write Control Sequence Logic-------------------------------------------------------------------------------
CASE Step_SEQ OF 					
	0:	// Enable Read & Write Logic
		IF xEnabled THEN 
			Lt_WriteIndex	:= 0;
			Step_SEQ		:= 10;
		ELSE
			Lt_WriteParaData[0].PreviousValue := 0;
            Lt_WriteParaData[1].PreviousValue := 0;
            Lt_WriteParaData[2].PreviousValue := 0;
            Lt_ReadParaData[0].Value := 0;
            xWriteDone := FALSE;
            Lt_WriteIndex := 0;
            Step_SEQ := 0;
		END_IF
	10:	// Read Data Parameter Input Logic 
		Lt_Read_Parameter_ISDU.Net_Id	        :=	sNetId ;
		Lt_Read_Parameter_ISDU.Ethercat_Address	:=	uiEthercatAddress ;
		Lt_Read_Parameter_ISDU.Slot_Number	    :=	uiSlotNumber ;
		Lt_Read_Parameter_ISDU.Port_Number		:=	usiPort;
		Lt_Read_Parameter_ISDU.Para_Index		:=	Lt_ReadParaData[Lt_ReadIndex].Index;
		Lt_Read_Parameter_ISDU.Para_SubIndex	:=	Lt_ReadParaData[Lt_ReadIndex].Sub_index;
		Lt_Read_Parameter_ISDU.Para_Length		:=	Lt_ReadParaData[Lt_ReadIndex].Length;
		(*Lt_Read_Parameter_ISDU.Para_Data[0]		:=	0;
		Lt_Read_Parameter_ISDU.Para_Data[1]		:=	0;
		Lt_Read_Parameter_ISDU.Para_Data[2]		:=	0;
		Lt_Read_Parameter_ISDU.Para_Data[3]		:=	0;*)
		
		Step_SEQ						:= 20;
		
	20:	// Read Command Enable Logic 
		
			Lt_Execute_Read		:=	TRUE;	 
		 	Step_SEQ			:= 21;
			
	21: // Read Feedback Data Manipulation
		IF ReadPara.xDone	THEN
			Lt_ReadParaData[0].Value	:= TO_DINT(Lt_Read_Parameter_ISDU.Para_Data[0]) + SHL(TO_DINT(Lt_Read_Parameter_ISDU.Para_Data[1]),8)	+ SHL(TO_DINT(Lt_Read_Parameter_ISDU.Para_Data[2]),16) 
														+ SHL(TO_DINT(Lt_Read_Parameter_ISDU.Para_Data[3]),24);
			Lt_Execute_Read					:= FALSE;
			Lt_WriteIndex := 0;
            Step_SEQ := 30;
		
			
		ELSIF	ReadPara.xError	THEN 
						
			Lt_Execute_Read					:= FALSE;
			Step_SEQ						:= 999;
			
		END_IF
	
	30: // Write Sequence	
		// Reset The Wrie ISDU Parameters Data
	
			Lt_Write_Parameter_ISDU.Para_Data[0]	:= 0;	
			Lt_Write_Parameter_ISDU.Para_Data[1]	:= 0;
			Lt_Write_Parameter_ISDU.Para_Data[2]	:= 0;
			Lt_Write_Parameter_ISDU.Para_Data[3]	:= 0;	
			Step_SEQ								:= 40;
			
	40:	// Write Data Parameter Input Logic 
		Lt_Write_Parameter_ISDU.Net_Id	:=	sNetId;
		Lt_Write_Parameter_ISDU.Ethercat_Address	:=	uiEthercatAddress;
		Lt_Write_Parameter_ISDU.Slot_Number	:=	uiSlotNumber;
		Lt_Write_Parameter_ISDU.Port_Number	:=	usiPort;
		Lt_Write_Parameter_ISDU.Para_Index	:=	Lt_WriteParaData[Lt_WriteIndex].Index;
		Lt_Write_Parameter_ISDU.Para_SubIndex	:=	Lt_WriteParaData[Lt_WriteIndex].Sub_index;
		Lt_Write_Parameter_ISDU.Para_Length		:=	Lt_WriteParaData[Lt_WriteIndex].Length;
		
		IF Lt_Write_Parameter_ISDU.Para_Length = 4 THEN
			
			Lt_RealConvert.rRealValue				:= Lt_WriteParaData[Lt_WriteIndex].REAL_Value;
			Lt_Write_Parameter_ISDU.Para_Data[0]	:= Lt_RealConvert.abyte[0];	
			Lt_Write_Parameter_ISDU.Para_Data[1]	:= Lt_RealConvert.abyte[1];
			Lt_Write_Parameter_ISDU.Para_Data[2]	:= Lt_RealConvert.abyte[2];
			Lt_Write_Parameter_ISDU.Para_Data[3]	:= Lt_RealConvert.abyte[3];	
		
		ELSIF Lt_Write_Parameter_ISDU.Para_Length = 2 THEN
			Lt_Write_Parameter_ISDU.Para_Data[0]	:=	TO_BYTE(Lt_WriteParaData[Lt_WriteIndex].Value);
			Lt_Write_Parameter_ISDU.Para_Data[1]	:=	TO_BYTE(SHR(Lt_WriteParaData[Lt_WriteIndex].Value,8));
		
		ELSIF Lt_Write_Parameter_ISDU.Para_Length = 1 THEN
			Lt_Write_Parameter_ISDU.Para_Data[0]	:=	TO_BYTE(Lt_WriteParaData[Lt_WriteIndex].Value);
		END_IF
			
		Step_SEQ						:= 50;
		
	50:	// Write Command Enable Logic 
		
            IF Lt_WriteParaData[Lt_WriteIndex].NeedAction THEN
				xWriteDone := FALSE;
                Lt_Execute_Write := TRUE;
                Step_SEQ := 60;
			ELSE
				Step_SEQ := 70;
            END_IF;
       		
	60:	// Write Data Manipulation
		IF WritePara.xDone THEN
			Lt_WriteParaData[Lt_WriteIndex].NeedAction		:= FALSE;
			Lt_WriteParaData[Lt_WriteIndex].PreviousValue	:= Lt_WriteParaData[Lt_WriteIndex].Value;
			Lt_Execute_Write								:= FALSE;
			xWriteDone										:= TRUE;
			Step_SEQ										:= 70;	 
		ELSIF WritePara.xError	THEN
			
			Lt_Execute_Write	:= FALSE;
			Step_SEQ			:= 999;
		 END_IF
	
	70:	// Write Parameter List Index & Move Sequence to Read Function Logic
		IF ( Lt_WriteIndex <= 2 ) THEN
	
			Lt_WriteIndex	:= Lt_WriteIndex + 1;
			Step_SEQ		:= 30;	
						
		ELSIF ( Lt_WriteIndex >= 3 ) THEN
			
			Step_SEQ		:= 10;
		END_IF	
	
	999:
		xError	:= TRUE;
						
END_CASE

ReadPara(
	xExecute:= Lt_Execute_Read, 
	sNetId:=Lt_Read_Parameter_ISDU.Net_Id , 
	uiEthercatAddress:=Lt_Read_Parameter_ISDU.Ethercat_Address , 
	uiSlotNumber:=Lt_Read_Parameter_ISDU.Slot_Number , 
	usiPort:=Lt_Read_Parameter_ISDU.Port_Number , 
	uiIndex:=Lt_Read_Parameter_ISDU.Para_Index , 
	usiSubIndex:=Lt_Read_Parameter_ISDU.Para_SubIndex , 
	pData:=ADR(Lt_Read_Parameter_ISDU.Para_Data[0]) , 
	uiDataLength:=Lt_Read_Parameter_ISDU.Para_Length , 
	xWrite:=FALSE , 
	xIsString:=Lt_IsItString , 
	xDone=> , 
	xBusy=> , 
	xError=> , 
	udiErrorCode=> , 
	eErrorDescription=> , 
	udiReadDataLength=> );
	
	WritePara(
	xExecute:=Lt_Execute_Write , 
	sNetId:=Lt_Write_Parameter_ISDU.Net_Id , 
	uiEthercatAddress:=Lt_Write_Parameter_ISDU.Ethercat_Address , 
	uiSlotNumber:=Lt_Write_Parameter_ISDU.Slot_Number , 
	usiPort:=Lt_Write_Parameter_ISDU.Port_Number , 
	uiIndex:=Lt_Write_Parameter_ISDU.Para_Index , 
	usiSubIndex:=Lt_Write_Parameter_ISDU.Para_SubIndex , 
	pData:=ADR(Lt_Write_Parameter_ISDU.Para_Data[0]) , 
	uiDataLength:=Lt_Write_Parameter_ISDU.Para_Length , 
	xWrite:=TRUE , 
	xIsString:=FALSE , 
	xDone=> , 
	xBusy=> , 
	xError=> , 
	udiErrorCode=> , 
	eErrorDescription=> , 
	udiReadDataLength=> );
				 
	// Current Position Feedback Value | Read Parameter Logic------------------------------------------------------------

diCurrentPosition           	:=  Lt_ReadParaData[0].Value;
Lt_ReadParaData[0].Sub_index	:= 16#0;
Lt_ReadParaData[0].Index		:= 16#120;
Lt_ReadParaData[0].Length		:= 4;

END_FUNCTION_BLOCK

// POUs/SMS_Festo_IO
FUNCTION_BLOCK SMS_Festo_IO
VAR_INPUT
	RefINPUTS: BYTE;
	xEnable: BOOL;
	xMoveIN: BOOL;
	xMoveIntermediate: BOOL;
	xMoveOut: BOOL;
	xQuitError: BOOL;
END_VAR
VAR_OUTPUT
	RefOUTPUTS: BYTE;
	xEnabled: BOOL;
	xStateIn: BOOL;
	xStateIntermediate: BOOL;
	xStateOut: BOOL;
	xStateMove: BOOL;
	xError: BOOL;
END_VAR
VAR
	Lt_StateDevice: BOOL;
END_VAR

(*
===============================================================================================================
Advice TO Released Library Revisions 
===============================================================================================================
SMS_Festo_Lib | Communication: Beckhoff EtherCat
---------------------------------------------------------------------------------------------------------------
Version                           Date of Release
V1.0                                07.01.2022
V1.1                                03.06.2022

---------------------------------------------------------------------------------------------------------------
Changes in Library:

V1.0 -  Release Version

*)
// Enable Function Block Sequence Logic------------------------------------------------------------------------ 
IF xEnable THEN 				
	xEnabled					:= TRUE;
	
ELSE
	xEnabled					:= FALSE;
	
END_IF

//Process Data Command Logic---------------------------------------------------------------------------------------
IF xEnabled THEN				
	
	IF xMoveIN THEN				// Move IN Position Command
		RefOUTPUTS.0	:= TRUE;
	ELSE
		RefOUTPUTS.0	:= FALSE;
	END_IF
	
	IF xMoveOut THEN			// Move OUT Position Command
		RefOUTPUTS.1	:= TRUE;
	ELSE
		RefOUTPUTS.1	:= FALSE;	
	END_IF
	
	IF xMoveIntermediate THEN	// Move Intermediat Position Command
		RefOUTPUTS.4	:= TRUE;
	ELSE
		RefOUTPUTS.4	:= FALSE;	
	END_IF
	
	IF xQuitError THEN			// Move Quite Error Command
		RefOUTPUTS.2	:= TRUE;
	ELSE
		RefOUTPUTS.2	:= FALSE;	
	END_IF
ELSE							// Clear Command When FB Not Enabled
	RefOUTPUTS.0	:= FALSE;	
	RefOUTPUTS.1	:= FALSE;	
	RefOUTPUTS.2	:= FALSE;
	RefOUTPUTS.4	:= FALSE;
END_IF


// Process Data Feedback Logic---------------------------------------------------------------------------------
IF xEnabled THEN				
	
	IF RefINPUTS.0 THEN				// IN Position Status
		xStateIn	:= TRUE;
	ELSE
		xStateIn	:= FALSE;
	END_IF
	
	IF RefINPUTS.1 THEN				// Out Position Status
		xStateOut	:= TRUE;
	ELSE
		xStateOut	:= FALSE;
	END_IF
	
	IF RefINPUTS.2 THEN				// Axis Moving Status
		xStateMove	:= TRUE;
	ELSE
		xStateMove	:= FALSE;
	END_IF
	
	IF RefINPUTS.3 THEN				// Device Healthy Status
		Lt_StateDevice	:= TRUE;
	ELSE
		Lt_StateDevice	:= FALSE;
	END_IF
	
	IF RefINPUTS.4 THEN				// Intermediat Position Status
		xStateIntermediate	:= TRUE;
	ELSE
		xStateIntermediate	:= FALSE;
	END_IF	
ELSE 								// Clear Status When FB is Not Enabled
	xStateIn			:= FALSE;
	xStateOut			:= FALSE;
	xStateMove			:= FALSE;
	xStateIntermediate	:= FALSE;
	Lt_StateDevice		:= FALSE;
END_IF

// Device Error State Logic -----------------------------------------------------------------------------------
IF xEnabled AND xStateIn AND xStateOut AND NOT Lt_StateDevice THEN
	xError	:= TRUE;
ELSE
	xError	:= FALSE;
END_IF

END_FUNCTION_BLOCK

// Project Information/F_GetCompany
// This function has been automatically generated from the project information.
{attribute 'signature_flag' := '1073741824'}
{attribute 'TcGenerated'}
{attribute 'no-analysis'}
FUNCTION F_GetCompany : WSTRING
VAR_INPUT
	
END_VAR

F_GetCompany := "Festo";

END_FUNCTION

// Project Information/F_GetTitle
// This function has been automatically generated from the project information.
{attribute 'signature_flag' := '1073741824'}
{attribute 'TcGenerated'}
{attribute 'no-analysis'}
FUNCTION F_GetTitle : WSTRING
VAR_INPUT
	
END_VAR

F_GetTitle := "SMS Festo Lib";

END_FUNCTION

// Project Information/F_GetVersion
// This function has been automatically generated from the project information.
{attribute 'signature_flag' := '1073741824'}
{attribute 'TcGenerated'}
{attribute 'no-analysis'}
FUNCTION F_GetVersion : ST_LibVersion
VAR_INPUT
	
END_VAR

F_GetVersion.iMajor := 1;
F_GetVersion.iMinor := 1;
F_GetVersion.iBuild := 0;
F_GetVersion.iRevision := 0;

END_FUNCTION
